LIN {X -0.269,Y -575.719,Z 1184.977,A 0.000,B 0.000,C 90.000,E1 31.799} C_DIS
LIN {X 0.203,Y -573.633,Z 1184.974,A 0.000,B 0.000,C 90.000,E1 31.209} C_DIS
LIN {X 0.086,Y -570.715,Z 1184.970,A 0.000,B 0.000,C 90.000,E1 30.541} C_DIS
LIN {X -0.150,Y -566.853,Z 1184.965,A 0.000,B 0.000,C 90.000,E1 29.745} C_DIS
LIN {X 0.163,Y -563.307,Z 1184.961,A 0.000,B 0.000,C 90.000,E1 29.027} C_DIS
LIN {X -0.358,Y -557.017,Z 1184.955,A 0.000,B 0.000,C 90.000,E1 27.975} C_DIS
LIN {X -0.139,Y -552.755,Z 1184.951,A 0.000,B 0.000,C 90.000,E1 27.257} C_DIS
LIN {X 0.150,Y -549.096,Z 1184.948,A 0.000,B 0.000,C 90.000,E1 26.668} C_DIS
LIN {X 0.138,Y -544.085,Z 1184.944,A 0.000,B 0.000,C 90.000,E1 25.976} C_DIS
LIN {X -0.009,Y -538.645,Z 1184.941,A 0.000,B 0.000,C 90.000,E1 25.283} C_DIS
LIN {X -0.197,Y -532.873,Z 1184.937,A 0.000,B 0.000,C 90.000,E1 24.591} C_DIS
LIN {X 0.108,Y -525.350,Z 1184.932,A 0.000,B 0.000,C 90.000,E1 23.695} C_DIS
LIN {X -0.102,Y -518.911,Z 1184.928,A 0.000,B 0.000,C 90.000,E1 23.003} C_DIS
LIN {X 0.115,Y -510.878,Z 1184.923,A 0.000,B 0.000,C 90.000,E1 22.153} C_DIS
LIN {X 0.130,Y -504.007,Z 1184.919,A 0.000,B 0.000,C 90.000,E1 21.461} C_DIS
LIN {X 0.176,Y -495.817,Z 1184.915,A 0.000,B 0.000,C 90.000,E1 20.663} C_DIS
LIN {X 0.012,Y -484.326,Z 1184.909,A 0.000,B 0.000,C 90.000,E1 19.631} C_DIS
LIN {X 0.204,Y -477.159,Z 1184.906,A 0.000,B 0.000,C 90.000,E1 18.960} C_DIS
LIN {X -0.109,Y -468.645,Z 1184.901,A 0.000,B 0.000,C 90.000,E1 18.236} C_DIS
LIN {X 0.094,Y -449.703,Z 1184.892,A 0.000,B 0.000,C 90.000,E1 16.496} C_DIS
LIN {X -0.072,Y -429.494,Z 1184.881,A 0.000,B 0.000,C 90.000,E1 14.537} C_DIS
LIN {X -0.024,Y -415.561,Z 1184.872,A 0.000,B 0.000,C 90.000,E1 13.008} C_DIS
LIN {X -0.139,Y -404.803,Z 1184.865,A 0.000,B 0.000,C 90.000,E1 11.715} C_DIS
LIN {X -0.011,Y -398.437,Z 1184.860,A 0.000,B 0.000,C 90.000,E1 10.838} C_DIS
LIN {X 0.029,Y -396.065,Z 1184.858,A 0.000,B 0.000,C 90.000,E1 10.433} C_DIS
LIN {X 0.074,Y -394.315,Z 1184.856,A 0.000,B 0.000,C 90.000,E1 10.074} C_DIS
LIN {X -0.105,Y -393.196,Z 1184.854,A 0.000,B 0.000,C 90.000,E1 9.792} C_DIS
LIN {X -0.142,Y -393.181,Z 1184.854,A 0.000,B 0.000,C 90.000,E1 9.792} C_DIS
LIN {X -0.065,Y -393.222,Z 1184.852,A 0.000,B 0.000,C 90.000,E1 9.443} C_DIS
LIN {X 0.077,Y -394.548,Z 1184.849,A 0.000,B 0.000,C 90.000,E1 8.803} C_DIS
LIN {X 0.005,Y -397.236,Z 1184.845,A 0.000,B 0.000,C 90.000,E1 8.106} C_DIS
LIN {X -0.079,Y -401.943,Z 1184.840,A 0.000,B 0.000,C 90.000,E1 7.239} C_DIS
LIN {X -0.159,Y -404.688,Z 1184.838,A 0.000,B 0.000,C 90.000,E1 6.891} C_DIS
LIN {X -0.150,Y -406.083,Z 1184.837,A 0.000,B 0.000,C 90.000,E1 6.720} C_DIS
LIN {X 0.070,Y -411.425,Z 1184.835,A 0.000,B 0.000,C 90.000,E1 6.201} C_DIS
LIN {X -0.139,Y -422.184,Z 1184.830,A 0.000,B 0.000,C 90.000,E1 5.391} C_DIS
LIN {X 0.231,Y -439.892,Z 1184.823,A 0.000,B 0.000,C 90.000,E1 4.012} C_DIS
LIN {X 0.057,Y -459.196,Z 1184.815,A 0.000,B 0.000,C 90.000,E1 2.636} C_DIS
LIN {X 0.128,Y -468.582,Z 1184.811,A 0.000,B 0.000,C 90.000,E1 1.949} C_DIS
LIN {X 0.139,Y -474.703,Z 1184.808,A 0.000,B 0.000,C 90.000,E1 1.489} C_DIS
LIN {X -0.061,Y -483.888,Z 1184.804,A 0.000,B 0.000,C 90.000,E1 0.802} C_DIS
LIN {X 0.030,Y -491.293,Z 1184.801,A 0.000,B 0.000,C 90.000,E1 0.172} C_DIS
LIN {X 0.065,Y -497.030,Z 1184.798,A 0.000,B 0.000,C 90.000,E1 359.656} C_DIS
LIN {X 0.152,Y -503.917,Z 1184.794,A 0.000,B 0.000,C 90.000,E1 358.969} C_DIS
LIN {X 0.242,Y -511.679,Z 1184.790,A 0.000,B 0.000,C 90.000,E1 358.108} C_DIS
LIN {X -0.203,Y -517.848,Z 1184.786,A 0.000,B 0.000,C 90.000,E1 357.421} C_DIS
LIN {X 0.215,Y -522.508,Z 1184.782,A 0.000,B 0.000,C 90.000,E1 356.788} C_DIS
LIN {X -0.165,Y -527.659,Z 1184.778,A 0.000,B 0.000,C 90.000,E1 356.102} C_DIS
LIN {X 0.060,Y -532.426,Z 1184.774,A 0.000,B 0.000,C 90.000,E1 355.355} C_DIS
LIN {X 0.070,Y -535.907,Z 1184.771,A 0.000,B 0.000,C 90.000,E1 354.780} C_DIS
LIN {X -0.108,Y -541.172,Z 1184.766,A 0.000,B 0.000,C 90.000,E1 353.799} C_DIS
LIN {X -0.034,Y -543.957,Z 1184.762,A 0.000,B 0.000,C 90.000,E1 353.223} C_DIS
LIN {X -0.132,Y -547.123,Z 1184.758,A 0.000,B 0.000,C 90.000,E1 352.527} C_DIS
LIN {X -0.279,Y -550.023,Z 1184.755,A 0.000,B 0.000,C 90.000,E1 351.837} C_DIS
LIN {X -0.041,Y -553.129,Z 1184.750,A 0.000,B 0.000,C 90.000,E1 350.971} C_DIS
LIN {X -0.225,Y -555.911,Z 1184.745,A 0.000,B 0.000,C 90.000,E1 350.151} C_DIS
LIN {X 0.212,Y -559.244,Z 1184.739,A 0.000,B 0.000,C 90.000,E1 348.993} C_DIS
LIN {X 0.097,Y -561.492,Z 1184.734,A 0.000,B 0.000,C 90.000,E1 348.173} C_DIS
LIN {X 0.167,Y -564.315,Z 1184.728,A 0.000,B 0.000,C 90.000,E1 347.061} C_DIS
LIN {X 0.025,Y -567.547,Z 1184.721,A 0.000,B 0.000,C 90.000,E1 345.700} C_DIS
LIN {X -0.058,Y -570.527,Z 1184.713,A 0.000,B 0.000,C 90.000,E1 344.338} C_DIS
LIN {X -0.281,Y -572.756,Z 1184.707,A 0.000,B 0.000,C 90.000,E1 343.268} C_DIS
LIN {X 0.055,Y -575.417,Z 1184.699,A 0.000,B 0.000,C 90.000,E1 341.873} C_DIS
LIN {X 0.075,Y -577.334,Z 1184.693,A 0.000,B 0.000,C 90.000,E1 340.786} C_DIS
LIN {X 0.115,Y -579.005,Z 1184.687,A 0.000,B 0.000,C 90.000,E1 339.699} C_DIS
LIN {X -0.163,Y -580.408,Z 1184.681,A 0.000,B 0.000,C 90.000,E1 338.646} C_DIS
LIN {X 0.264,Y -581.304,Z 1184.677,A 0.000,B 0.000,C 90.000,E1 337.794} C_DIS
LIN {X 0.015,Y -582.086,Z 1184.671,A 0.000,B 0.000,C 90.000,E1 336.741} C_DIS
LIN {X 0.142,Y -582.315,Z 1184.666,A 0.000,B 0.000,C 90.000,E1 335.921} C_DIS
LIN {X 0.275,Y -582.164,Z 1184.662,A 0.000,B 0.000,C 90.000,E1 335.101} C_DIS
LIN {X -0.119,Y -581.741,Z 1184.657,A 0.000,B 0.000,C 90.000,E1 334.332} C_DIS
LIN {X 0.008,Y -580.944,Z 1184.653,A 0.000,B 0.000,C 90.000,E1 333.512} C_DIS
LIN {X -0.261,Y -580.193,Z 1184.650,A 0.000,B 0.000,C 90.000,E1 332.999} C_DIS
LIN {X 0.108,Y -578.695,Z 1184.645,A 0.000,B 0.000,C 90.000,E1 332.153} C_DIS
LIN {X -0.321,Y -576.890,Z 1184.641,A 0.000,B 0.000,C 90.000,E1 331.385} C_DIS
LIN {X 0.163,Y -575.563,Z 1184.638,A 0.000,B 0.000,C 90.000,E1 330.795} C_DIS
LIN {X 0.137,Y -574.037,Z 1184.635,A 0.000,B 0.000,C 90.000,E1 330.255} C_DIS
LIN {X -0.183,Y -572.185,Z 1184.632,A 0.000,B 0.000,C 90.000,E1 329.744} C_DIS
LIN {X -0.059,Y -571.193,Z 1184.630,A 0.000,B 0.000,C 90.000,E1 329.459} C_DIS
LIN {X -0.108,Y -568.851,Z 1184.627,A 0.000,B 0.000,C 90.000,E1 328.918} C_DIS
LIN {X 0.106,Y -566.731,Z 1184.625,A 0.000,B 0.000,C 90.000,E1 328.486} C_DIS
LIN {X 0.018,Y -563.555,Z 1184.622,A 0.000,B 0.000,C 90.000,E1 327.946} C_DIS
LIN {X 0.106,Y -559.089,Z 1184.618,A 0.000,B 0.000,C 90.000,E1 327.248} C_DIS
LIN {X -0.033,Y -555.097,Z 1184.615,A 0.000,B 0.000,C 90.000,E1 326.707} C_DIS
LIN {X 0.108,Y -550.863,Z 1184.612,A 0.000,B 0.000,C 90.000,E1 326.135} C_DIS
LIN {X -0.220,Y -545.206,Z 1184.608,A 0.000,B 0.000,C 90.000,E1 325.468} C_DIS
LIN {X -0.265,Y -536.699,Z 1184.603,A 0.000,B 0.000,C 90.000,E1 324.482} C_DIS
LIN {X 0.122,Y -522.008,Z 1184.593,A 0.000,B 0.000,C 90.000,E1 322.763} C_DIS
LIN {X -0.102,Y -518.958,Z 1184.591,A 0.000,B 0.000,C 90.000,E1 322.351} C_DIS
LIN {X 0.324,Y -516.396,Z 1184.588,A 0.000,B 0.000,C 90.000,E1 321.823} C_DIS
LIN {X 0.010,Y -514.508,Z 1184.585,A 0.000,B 0.000,C 90.000,E1 321.251} C_DIS
LIN {X 0.113,Y -513.672,Z 1184.580,A 0.000,B 0.000,C 90.000,E1 320.356} C_DIS
LIN {X 0.035,Y -513.598,Z 1184.578,A 0.000,B 0.000,C 90.000,E1 320.070} C_DIS
LIN {X 0.125,Y -513.996,Z 1184.573,A 0.000,B 0.000,C 90.000,E1 319.175} C_DIS
LIN {X -0.168,Y -514.629,Z 1184.568,A 0.000,B 0.000,C 90.000,E1 318.324} C_DIS
LIN {X 0.079,Y -515.433,Z 1184.560,A 0.000,B 0.000,C 90.000,E1 316.824} C_DIS
LIN {X 0.163,Y -516.637,Z 1184.549,A 0.000,B 0.000,C 90.000,E1 314.757} C_DIS
LIN {X 0.077,Y -517.526,Z 1184.541,A 0.000,B 0.000,C 90.000,E1 313.299} C_DIS
LIN {X 0.236,Y -518.737,Z 1184.529,A 0.000,B 0.000,C 90.000,E1 311.229} C_DIS
LIN {X 0.147,Y -519.868,Z 1184.520,A 0.000,B 0.000,C 90.000,E1 309.483} C_DIS
LIN {X 0.150,Y -520.975,Z 1184.510,A 0.000,B 0.000,C 90.000,E1 307.729} C_DIS
LIN {X -0.141,Y -521.914,Z 1184.500,A 0.000,B 0.000,C 90.000,E1 306.011} C_DIS
LIN {X 0.052,Y -522.719,Z 1184.492,A 0.000,B 0.000,C 90.000,E1 304.532} C_DIS
LIN {X -0.084,Y -523.569,Z 1184.482,A 0.000,B 0.000,C 90.000,E1 302.801} C_DIS
LIN {X 0.002,Y -524.332,Z 1184.474,A 0.000,B 0.000,C 90.000,E1 301.337} C_DIS
LIN {X 0.029,Y -524.671,Z 1184.469,A 0.000,B 0.000,C 90.000,E1 300.463} C_DIS
LIN {X 0.138,Y -525.116,Z 1184.461,A 0.000,B 0.000,C 90.000,E1 298.999} C_DIS
LIN {X -0.007,Y -525.474,Z 1184.453,A 0.000,B 0.000,C 90.000,E1 297.564} C_DIS
LIN {X 0.082,Y -525.661,Z 1184.445,A 0.000,B 0.000,C 90.000,E1 296.104} C_DIS
LIN {X 0.180,Y -525.742,Z 1184.437,A 0.000,B 0.000,C 90.000,E1 294.643} C_DIS
LIN {X 0.062,Y -525.653,Z 1184.429,A 0.000,B 0.000,C 90.000,E1 293.206} C_DIS
LIN {X 0.106,Y -525.481,Z 1184.419,A 0.000,B 0.000,C 90.000,E1 291.461} C_DIS
LIN {X 0.269,Y -525.311,Z 1184.411,A 0.000,B 0.000,C 90.000,E1 289.993} C_DIS
LIN {X 0.089,Y -525.122,Z 1184.405,A 0.000,B 0.000,C 90.000,E1 288.852} C_DIS
LIN {X 0.077,Y -524.752,Z 1184.397,A 0.000,B 0.000,C 90.000,E1 287.402} C_DIS
LIN {X -0.099,Y -524.032,Z 1184.389,A 0.000,B 0.000,C 90.000,E1 285.969} C_DIS
LIN {X -0.149,Y -522.838,Z 1184.377,A 0.000,B 0.000,C 90.000,E1 283.939} C_DIS
LIN {X 0.007,Y -521.376,Z 1184.366,A 0.000,B 0.000,C 90.000,E1 281.883} C_DIS
LIN {X -0.078,Y -520.439,Z 1184.358,A 0.000,B 0.000,C 90.000,E1 280.433} C_DIS
LIN {X -0.081,Y -519.725,Z 1184.350,A 0.000,B 0.000,C 90.000,E1 278.973} C_DIS
LIN {X 0.244,Y -518.767,Z 1184.340,A 0.000,B 0.000,C 90.000,E1 277.182} C_DIS
LIN {X 0.049,Y -517.839,Z 1184.332,A 0.000,B 0.000,C 90.000,E1 275.739} C_DIS
LIN {X 0.131,Y -516.443,Z 1184.319,A 0.000,B 0.000,C 90.000,E1 273.383} C_DIS
LIN {X 0.140,Y -515.258,Z 1184.306,A 0.000,B 0.000,C 90.000,E1 271.031} C_DIS
LIN {X -0.140,Y -514.744,Z 1184.299,A 0.000,B 0.000,C 90.000,E1 269.885} C_DIS
LIN {X 0.011,Y -514.038,Z 1184.291,A 0.000,B 0.000,C 90.000,E1 268.396} C_DIS
LIN {X 0.158,Y -513.196,Z 1184.283,A 0.000,B 0.000,C 90.000,E1 266.906} C_DIS
LIN {X -0.193,Y -512.145,Z 1184.275,A 0.000,B 0.000,C 90.000,E1 265.469} C_DIS
LIN {X 0.043,Y -511.167,Z 1184.268,A 0.000,B 0.000,C 90.000,E1 264.261} C_DIS
LIN {X 0.218,Y -509.835,Z 1184.260,A 0.000,B 0.000,C 90.000,E1 262.761} C_DIS
LIN {X 0.221,Y -507.714,Z 1184.247,A 0.000,B 0.000,C 90.000,E1 260.387} C_DIS
LIN {X -0.110,Y -505.962,Z 1184.235,A 0.000,B 0.000,C 90.000,E1 258.342} C_DIS
LIN {X 0.057,Y -504.422,Z 1184.225,A 0.000,B 0.000,C 90.000,E1 256.533} C_DIS
LIN {X -0.007,Y -503.668,Z 1184.220,A 0.000,B 0.000,C 90.000,E1 255.644} C_DIS
LIN {X -0.080,Y -502.414,Z 1184.212,A 0.000,B 0.000,C 90.000,E1 254.157} C_DIS
LIN {X -0.045,Y -500.795,Z 1184.200,A 0.000,B 0.000,C 90.000,E1 252.054} C_DIS
LIN {X 0.041,Y -499.255,Z 1184.190,A 0.000,B 0.000,C 90.000,E1 250.242} C_DIS
LIN {X 0.189,Y -497.865,Z 1184.182,A 0.000,B 0.000,C 90.000,E1 248.720} C_DIS
LIN {X 0.084,Y -496.100,Z 1184.172,A 0.000,B 0.000,C 90.000,E1 246.922} C_DIS
LIN {X -0.162,Y -494.938,Z 1184.165,A 0.000,B 0.000,C 90.000,E1 245.741} C_DIS
LIN {X 0.031,Y -493.224,Z 1184.157,A 0.000,B 0.000,C 90.000,E1 244.204} C_DIS
LIN {X -0.054,Y -491.803,Z 1184.150,A 0.000,B 0.000,C 90.000,E1 242.999} C_DIS
LIN {X -0.106,Y -489.424,Z 1184.140,A 0.000,B 0.000,C 90.000,E1 241.179} C_DIS
LIN {X -0.033,Y -487.848,Z 1184.133,A 0.000,B 0.000,C 90.000,E1 239.950} C_DIS
LIN {X 0.067,Y -485.806,Z 1184.125,A 0.000,B 0.000,C 90.000,E1 238.408} C_DIS
LIN {X -0.279,Y -483.699,Z 1184.116,A 0.000,B 0.000,C 90.000,E1 236.914} C_DIS
LIN {X 0.295,Y -480.772,Z 1184.104,A 0.000,B 0.000,C 90.000,E1 234.689} C_DIS
LIN {X -0.078,Y -479.145,Z 1184.097,A 0.000,B 0.000,C 90.000,E1 233.497} C_DIS
LIN {X 0.079,Y -476.657,Z 1184.087,A 0.000,B 0.000,C 90.000,E1 231.618} C_DIS
LIN {X 0.015,Y -474.694,Z 1184.078,A 0.000,B 0.000,C 90.000,E1 230.070} C_DIS
LIN {X -0.137,Y -472.707,Z 1184.070,A 0.000,B 0.000,C 90.000,E1 228.528} C_DIS
LIN {X 0.082,Y -471.849,Z 1184.066,A 0.000,B 0.000,C 90.000,E1 227.877} C_DIS
LIN {X 0.003,Y -467.254,Z 1184.047,A 0.000,B 0.000,C 90.000,E1 224.433} C_DIS
LIN {X 0.157,Y -464.953,Z 1184.035,A 0.000,B 0.000,C 90.000,E1 222.204} C_DIS
LIN {X -0.172,Y -463.095,Z 1184.010,A 0.000,B 0.000,C 90.000,E1 217.810} C_DIS
LIN {X -0.268,Y -463.009,Z 1184.005,A 0.000,B 0.000,C 90.000,E1 216.870} C_DIS
LIN {X 0.030,Y -462.884,Z 1183.992,A 0.000,B 0.000,C 90.000,E1 214.612} C_DIS
LIN {X -0.057,Y -463.639,Z 1183.978,A 0.000,B 0.000,C 90.000,E1 212.084} C_DIS
LIN {X -0.248,Y -465.015,Z 1183.968,A 0.000,B 0.000,C 90.000,E1 210.207} C_DIS
LIN {X -0.010,Y -467.601,Z 1183.952,A 0.000,B 0.000,C 90.000,E1 207.334} C_DIS
LIN {X -0.234,Y -474.700,Z 1183.922,A 0.000,B 0.000,C 90.000,E1 202.025} C_DIS
LIN {X 0.287,Y -482.358,Z 1183.901,A 0.000,B 0.000,C 90.000,E1 198.236} C_DIS
LIN {X -0.133,Y -493.316,Z 1183.879,A 0.000,B 0.000,C 90.000,E1 194.300} C_DIS
LIN {X -0.074,Y -499.996,Z 1183.868,A 0.000,B 0.000,C 90.000,E1 192.175} C_DIS
LIN {X 0.000,Y -505.831,Z 1183.858,A 0.000,B 0.000,C 90.000,E1 190.366} C_DIS
LIN {X 0.124,Y -511.908,Z 1183.848,A 0.000,B 0.000,C 90.000,E1 188.568} C_DIS
LIN {X -0.175,Y -516.997,Z 1183.839,A 0.000,B 0.000,C 90.000,E1 187.125} C_DIS
LIN {X 0.138,Y -521.938,Z 1183.831,A 0.000,B 0.000,C 90.000,E1 185.625} C_DIS
LIN {X -0.063,Y -528.889,Z 1183.820,A 0.000,B 0.000,C 90.000,E1 183.612} C_DIS
LIN {X -0.138,Y -533.797,Z 1183.812,A 0.000,B 0.000,C 90.000,E1 182.178} C_DIS
LIN {X -0.132,Y -537.755,Z 1183.806,A 0.000,B 0.000,C 90.000,E1 181.031} C_DIS
LIN {X -0.006,Y -544.608,Z 1183.795,A 0.000,B 0.000,C 90.000,E1 179.026} C_DIS
LIN {X 0.206,Y -549.498,Z 1183.787,A 0.000,B 0.000,C 90.000,E1 177.593} C_DIS
LIN {X -0.045,Y -554.277,Z 1183.779,A 0.000,B 0.000,C 90.000,E1 176.216} C_DIS
LIN {X -0.181,Y -559.046,Z 1183.771,A 0.000,B 0.000,C 90.000,E1 174.837} C_DIS
LIN {X 0.067,Y -565.560,Z 1183.760,A 0.000,B 0.000,C 90.000,E1 172.875} C_DIS
LIN {X 0.196,Y -570.165,Z 1183.753,A 0.000,B 0.000,C 90.000,E1 171.489} C_DIS
LIN {X -0.274,Y -573.811,Z 1183.747,A 0.000,B 0.000,C 90.000,E1 170.443} C_DIS
LIN {X 0.080,Y -578.337,Z 1183.739,A 0.000,B 0.000,C 90.000,E1 169.050} C_DIS
LIN {X 0.289,Y -583.650,Z 1183.730,A 0.000,B 0.000,C 90.000,E1 167.409} C_DIS
LIN {X -0.214,Y -588.094,Z 1183.723,A 0.000,B 0.000,C 90.000,E1 166.117} C_DIS
LIN {X 0.069,Y -592.417,Z 1183.715,A 0.000,B 0.000,C 90.000,E1 164.755} C_DIS
LIN {X 0.298,Y -597.572,Z 1183.707,A 0.000,B 0.000,C 90.000,E1 163.142} C_DIS
LIN {X -0.123,Y -600.956,Z 1183.701,A 0.000,B 0.000,C 90.000,E1 162.127} C_DIS
LIN {X 0.256,Y -604.285,Z 1183.695,A 0.000,B 0.000,C 90.000,E1 161.040} C_DIS
LIN {X 0.043,Y -608.346,Z 1183.688,A 0.000,B 0.000,C 90.000,E1 159.752} C_DIS
LIN {X -0.049,Y -611.504,Z 1183.682,A 0.000,B 0.000,C 90.000,E1 158.720} C_DIS
LIN {X 0.088,Y -615.385,Z 1183.675,A 0.000,B 0.000,C 90.000,E1 157.411} C_DIS
LIN {X 0.317,Y -618.494,Z 1183.669,A 0.000,B 0.000,C 90.000,E1 156.357} C_DIS
LIN {X 0.016,Y -621.525,Z 1183.663,A 0.000,B 0.000,C 90.000,E1 155.357} C_DIS
LIN {X 0.034,Y -625.811,Z 1183.655,A 0.000,B 0.000,C 90.000,E1 153.819} C_DIS
LIN {X 0.122,Y -629.295,Z 1183.648,A 0.000,B 0.000,C 90.000,E1 152.538} C_DIS
LIN {X 0.259,Y -632.697,Z 1183.641,A 0.000,B 0.000,C 90.000,E1 151.257} C_DIS
LIN {X 0.157,Y -635.267,Z 1183.635,A 0.000,B 0.000,C 90.000,E1 150.255} C_DIS
LIN {X -0.229,Y -637.787,Z 1183.629,A 0.000,B 0.000,C 90.000,E1 149.282} C_DIS
LIN {X 0.122,Y -640.675,Z 1183.622,A 0.000,B 0.000,C 90.000,E1 147.995} C_DIS
LIN {X 0.123,Y -642.870,Z 1183.617,A 0.000,B 0.000,C 90.000,E1 146.993} C_DIS
LIN {X -0.034,Y -644.980,Z 1183.611,A 0.000,B 0.000,C 90.000,E1 146.008} C_DIS
LIN {X -0.102,Y -647.422,Z 1183.604,A 0.000,B 0.000,C 90.000,E1 144.769} C_DIS
LIN {X 0.154,Y -650.152,Z 1183.596,A 0.000,B 0.000,C 90.000,E1 143.256} C_DIS
LIN {X 0.072,Y -652.762,Z 1183.588,A 0.000,B 0.000,C 90.000,E1 141.778} C_DIS
LIN {X -0.180,Y -656.501,Z 1183.577,A 0.000,B 0.000,C 90.000,E1 139.828} C_DIS
LIN {X -0.265,Y -658.488,Z 1183.571,A 0.000,B 0.000,C 90.000,E1 138.852} C_DIS
LIN {X 0.090,Y -661.172,Z 1183.564,A 0.000,B 0.000,C 90.000,E1 137.595} C_DIS
LIN {X 0.031,Y -664.270,Z 1183.556,A 0.000,B 0.000,C 90.000,E1 136.134} C_DIS
LIN {X 0.011,Y -668.494,Z 1183.546,A 0.000,B 0.000,C 90.000,E1 134.190} C_DIS
LIN {X 0.162,Y -674.179,Z 1183.532,A 0.000,B 0.000,C 90.000,E1 131.757} C_DIS
LIN {X -0.441,Y -679.395,Z 1183.520,A 0.000,B 0.000,C 90.000,E1 129.644} C_DIS
LIN {X -0.060,Y -682.953,Z 1183.512,A 0.000,B 0.000,C 90.000,E1 128.177} C_DIS
LIN {X -0.366,Y -687.741,Z 1183.502,A 0.000,B 0.000,C 90.000,E1 126.297} C_DIS
LIN {X -0.285,Y -690.679,Z 1183.495,A 0.000,B 0.000,C 90.000,E1 125.105} C_DIS
LIN {X -0.158,Y -693.453,Z 1183.488,A 0.000,B 0.000,C 90.000,E1 123.913} C_DIS
LIN {X -0.027,Y -695.531,Z 1183.483,A 0.000,B 0.000,C 90.000,E1 122.959} C_DIS
LIN {X -0.213,Y -698.049,Z 1183.477,A 0.000,B 0.000,C 90.000,E1 121.799} C_DIS
LIN {X 0.232,Y -700.396,Z 1183.470,A 0.000,B 0.000,C 90.000,E1 120.590} C_DIS
LIN {X -0.249,Y -702.441,Z 1183.464,A 0.000,B 0.000,C 90.000,E1 119.461} C_DIS
LIN {X 0.245,Y -703.928,Z 1183.458,A 0.000,B 0.000,C 90.000,E1 118.487} C_DIS
LIN {X -0.188,Y -705.309,Z 1183.453,A 0.000,B 0.000,C 90.000,E1 117.590} C_DIS
LIN {X 0.056,Y -706.086,Z 1183.449,A 0.000,B 0.000,C 90.000,E1 116.873} C_DIS
LIN {X -0.351,Y -706.587,Z 1183.444,A 0.000,B 0.000,C 90.000,E1 115.976} C_DIS
LIN {X 0.238,Y -706.682,Z 1183.442,A 0.000,B 0.000,C 90.000,E1 115.463} C_DIS
LIN {X 0.179,Y -706.508,Z 1183.438,A 0.000,B 0.000,C 90.000,E1 114.771} C_DIS
LIN {X -0.171,Y -706.409,Z 1183.436,A 0.000,B 0.000,C 90.000,E1 114.567} C_DIS
LIN {X 0.120,Y -705.564,Z 1183.434,A 0.000,B 0.000,C 90.000,E1 114.079} C_DIS
LIN {X 0.410,Y -704.995,Z 1183.433,A 0.000,B 0.000,C 90.000,E1 113.823} C_DIS
LIN {X 0.052,Y -702.907,Z 1183.430,A 0.000,B 0.000,C 90.000,E1 113.387} C_DIS
LIN {X 0.190,Y -702.299,Z 1183.429,A 0.000,B 0.000,C 90.000,E1 113.259} C_DIS
LIN {X 0.053,Y -701.383,Z 1183.429,A 0.000,B 0.000,C 90.000,E1 113.153} C_DIS
LIN {X 0.035,Y -696.336,Z 1183.426,A 0.000,B 0.000,C 90.000,E1 112.695} C_DIS
LIN {X -0.031,Y -694.686,Z 1183.426,A 0.000,B 0.000,C 90.000,E1 112.589} C_DIS
LIN {X 0.171,Y -691.695,Z 1183.425,A 0.000,B 0.000,C 90.000,E1 112.461} C_DIS
LIN {X 0.102,Y -685.305,Z 1183.424,A 0.000,B 0.000,C 90.000,E1 112.280} C_DIS
LIN {X -0.112,Y -683.759,Z 1183.424,A 0.000,B 0.000,C 90.000,E1 112.280} C_DIS
LIN {X -0.109,Y -677.261,Z 1183.424,A 0.000,B 0.000,C 90.000,E1 112.259} C_DIS
LIN {X -0.142,Y -606.123,Z 1183.424,A 0.000,B 0.000,C 90.000,E1 112.259} C_DIS
LIN {X -0.123,Y -601.588,Z 1183.422,A 0.000,B 0.000,C 90.000,E1 111.950} C_DIS
LIN {X -0.165,Y -590.164,Z 1183.417,A 0.000,B 0.000,C 90.000,E1 111.025} C_DIS
LIN {X -0.077,Y -578.973,Z 1183.412,A 0.000,B 0.000,C 90.000,E1 110.120} C_DIS
LIN {X -0.012,Y -569.965,Z 1183.408,A 0.000,B 0.000,C 90.000,E1 109.450} C_DIS
LIN {X 0.012,Y -556.759,Z 1183.403,A 0.000,B 0.000,C 90.000,E1 108.489} C_DIS
LIN {X 0.021,Y -553.886,Z 1183.401,A 0.000,B 0.000,C 90.000,E1 108.181} C_DIS
LIN {X -0.107,Y -553.394,Z 1183.401,A 0.000,B 0.000,C 90.000,E1 108.127} C_DIS
LIN {X 0.212,Y -552.038,Z 1183.399,A 0.000,B 0.000,C 90.000,E1 107.819} C_DIS
LIN {X 0.187,Y -551.203,Z 1183.397,A 0.000,B 0.000,C 90.000,E1 107.402} C_DIS
LIN {X 0.026,Y -550.969,Z 1183.394,A 0.000,B 0.000,C 90.000,E1 106.858} C_DIS
LIN {X -0.036,Y -551.484,Z 1183.389,A 0.000,B 0.000,C 90.000,E1 106.024} C_DIS
LIN {X -0.146,Y -552.999,Z 1183.380,A 0.000,B 0.000,C 90.000,E1 104.356} C_DIS
LIN {X -0.122,Y -554.806,Z 1183.367,A 0.000,B 0.000,C 90.000,E1 102.119} C_DIS
LIN {X 0.144,Y -556.784,Z 1183.356,A 0.000,B 0.000,C 90.000,E1 100.141} C_DIS
LIN {X 0.188,Y -558.293,Z 1183.349,A 0.000,B 0.000,C 90.000,E1 98.746} C_DIS
LIN {X 0.251,Y -559.627,Z 1183.341,A 0.000,B 0.000,C 90.000,E1 97.352} C_DIS
LIN {X 0.117,Y -560.543,Z 1183.335,A 0.000,B 0.000,C 90.000,E1 96.258} C_DIS
LIN {X 0.218,Y -561.694,Z 1183.326,A 0.000,B 0.000,C 90.000,E1 94.588} C_DIS
LIN {X -0.268,Y -562.787,Z 1183.316,A 0.000,B 0.000,C 90.000,E1 92.980} C_DIS
LIN {X -0.092,Y -564.228,Z 1183.306,A 0.000,B 0.000,C 90.000,E1 91.031} C_DIS
LIN {X 0.001,Y -565.456,Z 1183.297,A 0.000,B 0.000,C 90.000,E1 89.370} C_DIS
LIN {X 0.133,Y -566.581,Z 1183.287,A 0.000,B 0.000,C 90.000,E1 87.707} C_DIS
LIN {X -0.282,Y -567.721,Z 1183.278,A 0.000,B 0.000,C 90.000,E1 86.102} C_DIS
LIN {X -0.194,Y -568.668,Z 1183.271,A 0.000,B 0.000,C 90.000,E1 84.723} C_DIS
LIN {X 0.080,Y -569.811,Z 1183.261,A 0.000,B 0.000,C 90.000,E1 83.053} C_DIS
LIN {X -0.302,Y -570.711,Z 1183.254,A 0.000,B 0.000,C 90.000,E1 81.724} C_DIS
LIN {X -0.210,Y -571.384,Z 1183.248,A 0.000,B 0.000,C 90.000,E1 80.622} C_DIS
LIN {X 0.188,Y -572.174,Z 1183.240,A 0.000,B 0.000,C 90.000,E1 79.218} C_DIS
LIN {X -0.235,Y -573.206,Z 1183.230,A 0.000,B 0.000,C 90.000,E1 77.353} C_DIS
LIN {X -0.031,Y -574.064,Z 1183.221,A 0.000,B 0.000,C 90.000,E1 75.700} C_DIS
LIN {X 0.187,Y -574.886,Z 1183.212,A 0.000,B 0.000,C 90.000,E1 74.047} C_DIS
LIN {X -0.158,Y -576.247,Z 1183.198,A 0.000,B 0.000,C 90.000,E1 71.638} C_DIS
LIN {X 0.257,Y -577.413,Z 1183.187,A 0.000,B 0.000,C 90.000,E1 69.699} C_DIS
LIN {X 0.209,Y -579.237,Z 1183.175,A 0.000,B 0.000,C 90.000,E1 67.539} C_DIS
LIN {X 0.185,Y -580.912,Z 1183.166,A 0.000,B 0.000,C 90.000,E1 65.921} C_DIS
LIN {X 0.297,Y -582.639,Z 1183.156,A 0.000,B 0.000,C 90.000,E1 64.024} C_DIS
LIN {X 0.189,Y -584.506,Z 1183.146,A 0.000,B 0.000,C 90.000,E1 62.153} C_DIS
LIN {X -0.271,Y -585.991,Z 1183.136,A 0.000,B 0.000,C 90.000,E1 60.589} C_DIS
LIN {X 0.087,Y -587.390,Z 1183.128,A 0.000,B 0.000,C 90.000,E1 58.948} C_DIS
LIN {X 0.204,Y -588.233,Z 1183.122,A 0.000,B 0.000,C 90.000,E1 57.867} C_DIS
LIN {X 0.037,Y -589.178,Z 1183.114,A 0.000,B 0.000,C 90.000,E1 56.548} C_DIS
LIN {X -0.105,Y -590.148,Z 1183.107,A 0.000,B 0.000,C 90.000,E1 55.229} C_DIS
LIN {X 0.036,Y -590.900,Z 1183.101,A 0.000,B 0.000,C 90.000,E1 54.149} C_DIS
LIN {X 0.186,Y -591.535,Z 1183.096,A 0.000,B 0.000,C 90.000,E1 53.336} C_DIS
LIN {X -0.025,Y -593.012,Z 1183.083,A 0.000,B 0.000,C 90.000,E1 50.964} C_DIS
LIN {X 0.129,Y -593.608,Z 1183.076,A 0.000,B 0.000,C 90.000,E1 49.622} C_DIS
LIN {X 0.055,Y -594.283,Z 1183.067,A 0.000,B 0.000,C 90.000,E1 48.038} C_DIS
LIN {X -0.028,Y -594.459,Z 1183.061,A 0.000,B 0.000,C 90.000,E1 46.986} C_DIS
LIN {X -0.122,Y -594.491,Z 1183.052,A 0.000,B 0.000,C 90.000,E1 45.405} C_DIS
LIN {X -0.189,Y -594.320,Z 1183.046,A 0.000,B 0.000,C 90.000,E1 44.352} C_DIS
LIN {X -0.033,Y -594.046,Z 1183.042,A 0.000,B 0.000,C 90.000,E1 43.542} C_DIS
LIN {X -0.290,Y -593.608,Z 1183.037,A 0.000,B 0.000,C 90.000,E1 42.771} C_DIS
LIN {X -0.181,Y -592.733,Z 1183.030,A 0.000,B 0.000,C 90.000,E1 41.434} C_DIS
LIN {X -0.003,Y -592.182,Z 1183.026,A 0.000,B 0.000,C 90.000,E1 40.620} C_DIS
LIN {X 0.135,Y -590.914,Z 1183.018,A 0.000,B 0.000,C 90.000,E1 39.277} C_DIS
LIN {X 0.041,Y -589.797,Z 1183.012,A 0.000,B 0.000,C 90.000,E1 38.222} C_DIS
LIN {X 0.088,Y -589.128,Z 1183.009,A 0.000,B 0.000,C 90.000,E1 37.684} C_DIS
LIN {X -0.196,Y -587.049,Z 1183.002,A 0.000,B 0.000,C 90.000,E1 36.377} C_DIS
LIN {X -0.240,Y -585.137,Z 1182.996,A 0.000,B 0.000,C 90.000,E1 35.311} C_DIS
LIN {X 0.132,Y -583.973,Z 1182.993,A 0.000,B 0.000,C 90.000,E1 34.739} C_DIS
LIN {X -0.293,Y -581.353,Z 1182.987,A 0.000,B 0.000,C 90.000,E1 33.706} C_DIS
LIN {X -0.264,Y -578.121,Z 1182.981,A 0.000,B 0.000,C 90.000,E1 32.625} C_DIS
LIN {X -0.117,Y -575.306,Z 1182.977,A 0.000,B 0.000,C 90.000,E1 31.799} C_DIS
LIN {X -0.140,Y -573.231,Z 1182.974,A 0.000,B 0.000,C 90.000,E1 31.258} C_DIS
LIN {X -0.262,Y -570.273,Z 1182.970,A 0.000,B 0.000,C 90.000,E1 30.590} C_DIS
LIN {X -0.102,Y -565.727,Z 1182.964,A 0.000,B 0.000,C 90.000,E1 29.617} C_DIS
LIN {X -0.293,Y -562.104,Z 1182.961,A 0.000,B 0.000,C 90.000,E1 28.949} C_DIS
LIN {X -0.337,Y -555.728,Z 1182.955,A 0.000,B 0.000,C 90.000,E1 27.847} C_DIS
LIN {X -0.130,Y -551.354,Z 1182.951,A 0.000,B 0.000,C 90.000,E1 27.129} C_DIS
LIN {X 0.019,Y -548.594,Z 1182.948,A 0.000,B 0.000,C 90.000,E1 26.693} C_DIS
LIN {X 0.048,Y -542.411,Z 1182.944,A 0.000,B 0.000,C 90.000,E1 25.848} C_DIS
LIN {X -0.091,Y -536.952,Z 1182.940,A 0.000,B 0.000,C 90.000,E1 25.155} C_DIS
LIN {X -0.296,Y -531.006,Z 1182.936,A 0.000,B 0.000,C 90.000,E1 24.463} C_DIS
LIN {X -0.154,Y -522.173,Z 1182.930,A 0.000,B 0.000,C 90.000,E1 23.439} C_DIS
LIN {X 0.256,Y -516.872,Z 1182.927,A 0.000,B 0.000,C 90.000,E1 22.823} C_DIS
LIN {X -0.042,Y -507.536,Z 1182.922,A 0.000,B 0.000,C 90.000,E1 21.897} C_DIS
LIN {X 0.071,Y -496.324,Z 1182.916,A 0.000,B 0.000,C 90.000,E1 20.791} C_DIS
LIN {X -0.159,Y -484.736,Z 1182.910,A 0.000,B 0.000,C 90.000,E1 19.758} C_DIS
LIN {X -0.108,Y -477.357,Z 1182.906,A 0.000,B 0.000,C 90.000,E1 19.087} C_DIS
LIN {X -0.174,Y -468.548,Z 1182.902,A 0.000,B 0.000,C 90.000,E1 18.308} C_DIS
LIN {X 0.130,Y -448.451,Z 1182.891,A 0.000,B 0.000,C 90.000,E1 16.441} C_DIS
LIN {X 0.090,Y -429.593,Z 1182.881,A 0.000,B 0.000,C 90.000,E1 14.592} C_DIS
LIN {X 0.036,Y -415.515,Z 1182.873,A 0.000,B 0.000,C 90.000,E1 13.063} C_DIS
LIN {X 0.179,Y -404.697,Z 1182.865,A 0.000,B 0.000,C 90.000,E1 11.715} C_DIS
LIN {X -0.167,Y -398.247,Z 1182.860,A 0.000,B 0.000,C 90.000,E1 10.894} C_DIS
LIN {X -0.158,Y -395.251,Z 1182.858,A 0.000,B 0.000,C 90.000,E1 10.366} C_DIS
LIN {X -0.205,Y -394.427,Z 1182.857,A 0.000,B 0.000,C 90.000,E1 10.197} C_DIS
LIN {X -0.115,Y -393.206,Z 1182.855,A 0.000,B 0.000,C 90.000,E1 9.849} C_DIS
LIN {X -0.153,Y -393.197,Z 1182.855,A 0.000,B 0.000,C 90.000,E1 9.849} C_DIS
LIN {X -0.067,Y -393.253,Z 1182.852,A 0.000,B 0.000,C 90.000,E1 9.443} C_DIS
LIN {X -0.096,Y -394.427,Z 1182.849,A 0.000,B 0.000,C 90.000,E1 8.916} C_DIS
LIN {X -0.135,Y -395.593,Z 1182.848,A 0.000,B 0.000,C 90.000,E1 8.568} C_DIS
LIN {X 0.180,Y -397.641,Z 1182.845,A 0.000,B 0.000,C 90.000,E1 7.992} C_DIS
LIN {X 0.102,Y -402.314,Z 1182.840,A 0.000,B 0.000,C 90.000,E1 7.125} C_DIS
LIN {X 0.107,Y -406.480,Z 1182.837,A 0.000,B 0.000,C 90.000,E1 6.606} C_DIS
LIN {X -0.058,Y -411.855,Z 1182.834,A 0.000,B 0.000,C 90.000,E1 6.144} C_DIS
LIN {X 0.021,Y -421.410,Z 1182.830,A 0.000,B 0.000,C 90.000,E1 5.391} C_DIS
LIN {X -0.100,Y -440.743,Z 1182.822,A 0.000,B 0.000,C 90.000,E1 3.955} C_DIS
LIN {X -0.102,Y -459.811,Z 1182.814,A 0.000,B 0.000,C 90.000,E1 2.579} C_DIS
LIN {X -0.050,Y -470.866,Z 1182.810,A 0.000,B 0.000,C 90.000,E1 1.776} C_DIS
LIN {X -0.212,Y -481.583,Z 1182.805,A 0.000,B 0.000,C 90.000,E1 0.974} C_DIS
LIN {X 0.078,Y -487.546,Z 1182.803,A 0.000,B 0.000,C 90.000,E1 0.458} C_DIS
LIN {X -0.140,Y -491.931,Z 1182.801,A 0.000,B 0.000,C 90.000,E1 0.115} C_DIS
LIN {X 0.064,Y -496.865,Z 1182.798,A 0.000,B 0.000,C 90.000,E1 359.656} C_DIS
LIN {X 0.164,Y -503.823,Z 1182.794,A 0.000,B 0.000,C 90.000,E1 358.969} C_DIS
LIN {X -0.190,Y -511.596,Z 1182.790,A 0.000,B 0.000,C 90.000,E1 358.165} C_DIS
LIN {X -0.092,Y -517.785,Z 1182.786,A 0.000,B 0.000,C 90.000,E1 357.421} C_DIS
LIN {X -0.160,Y -522.458,Z 1182.782,A 0.000,B 0.000,C 90.000,E1 356.846} C_DIS
LIN {X -0.265,Y -528.617,Z 1182.778,A 0.000,B 0.000,C 90.000,E1 355.988} C_DIS
LIN {X 0.243,Y -532.449,Z 1182.774,A 0.000,B 0.000,C 90.000,E1 355.355} C_DIS
LIN {X 0.254,Y -535.967,Z 1182.771,A 0.000,B 0.000,C 90.000,E1 354.780} C_DIS
LIN {X -0.191,Y -540.565,Z 1182.766,A 0.000,B 0.000,C 90.000,E1 353.970} C_DIS
LIN {X -0.120,Y -543.446,Z 1182.763,A 0.000,B 0.000,C 90.000,E1 353.394} C_DIS
LIN {X 0.251,Y -546.690,Z 1182.759,A 0.000,B 0.000,C 90.000,E1 352.648} C_DIS
LIN {X -0.084,Y -550.237,Z 1182.755,A 0.000,B 0.000,C 90.000,E1 351.837} C_DIS
LIN {X 0.157,Y -553.353,Z 1182.750,A 0.000,B 0.000,C 90.000,E1 350.971} C_DIS
LIN {X -0.025,Y -556.153,Z 1182.745,A 0.000,B 0.000,C 90.000,E1 350.151} C_DIS
LIN {X -0.132,Y -559.510,Z 1182.739,A 0.000,B 0.000,C 90.000,E1 349.050} C_DIS
LIN {X -0.091,Y -562.530,Z 1182.733,A 0.000,B 0.000,C 90.000,E1 347.937} C_DIS
LIN {X -0.007,Y -565.290,Z 1182.727,A 0.000,B 0.000,C 90.000,E1 346.825} C_DIS
LIN {X -0.131,Y -568.501,Z 1182.719,A 0.000,B 0.000,C 90.000,E1 345.463} C_DIS
LIN {X -0.200,Y -571.434,Z 1182.712,A 0.000,B 0.000,C 90.000,E1 344.102} C_DIS
LIN {X 0.303,Y -573.643,Z 1182.706,A 0.000,B 0.000,C 90.000,E1 342.960} C_DIS
LIN {X -0.064,Y -576.296,Z 1182.698,A 0.000,B 0.000,C 90.000,E1 341.638} C_DIS
LIN {X -0.037,Y -578.192,Z 1182.692,A 0.000,B 0.000,C 90.000,E1 340.550} C_DIS
LIN {X 0.214,Y -579.817,Z 1182.686,A 0.000,B 0.000,C 90.000,E1 339.444} C_DIS
LIN {X 0.098,Y -580.889,Z 1182.682,A 0.000,B 0.000,C 90.000,E1 338.646} C_DIS
LIN {X -0.150,Y -582.072,Z 1182.676,A 0.000,B 0.000,C 90.000,E1 337.592} C_DIS
LIN {X 0.153,Y -582.737,Z 1182.670,A 0.000,B 0.000,C 90.000,E1 336.485} C_DIS
LIN {X -0.110,Y -582.898,Z 1182.667,A 0.000,B 0.000,C 90.000,E1 335.973} C_DIS
LIN {X 0.161,Y -582.890,Z 1182.664,A 0.000,B 0.000,C 90.000,E1 335.409} C_DIS
LIN {X 0.302,Y -582.549,Z 1182.659,A 0.000,B 0.000,C 90.000,E1 334.588} C_DIS
LIN {X -0.086,Y -581.894,Z 1182.655,A 0.000,B 0.000,C 90.000,E1 333.819} C_DIS
LIN {X 0.173,Y -581.336,Z 1182.652,A 0.000,B 0.000,C 90.000,E1 333.256} C_DIS
LIN {X -0.229,Y -580.011,Z 1182.647,A 0.000,B 0.000,C 90.000,E1 332.487} C_DIS
LIN {X 0.139,Y -578.344,Z 1182.643,A 0.000,B 0.000,C 90.000,E1 331.641} C_DIS
LIN {X -0.019,Y -576.421,Z 1182.638,A 0.000,B 0.000,C 90.000,E1 330.845} C_DIS
LIN {X 0.307,Y -574.103,Z 1182.634,A 0.000,B 0.000,C 90.000,E1 329.999} C_DIS
LIN {X 0.108,Y -571.063,Z 1182.629,A 0.000,B 0.000,C 90.000,E1 329.203} C_DIS
LIN {X 0.143,Y -569.234,Z 1182.627,A 0.000,B 0.000,C 90.000,E1 328.791} C_DIS
LIN {X -0.126,Y -567.087,Z 1182.625,A 0.000,B 0.000,C 90.000,E1 328.408} C_DIS
LIN {X -0.007,Y -563.004,Z 1182.621,A 0.000,B 0.000,C 90.000,E1 327.709} C_DIS
LIN {X -0.009,Y -560.398,Z 1182.618,A 0.000,B 0.000,C 90.000,E1 327.296} C_DIS
LIN {X -0.361,Y -554.367,Z 1182.614,A 0.000,B 0.000,C 90.000,E1 326.501} C_DIS
LIN {X 0.356,Y -551.194,Z 1182.611,A 0.000,B 0.000,C 90.000,E1 326.008} C_DIS
LIN {X 0.159,Y -546.622,Z 1182.608,A 0.000,B 0.000,C 90.000,E1 325.468} C_DIS
LIN {X 0.125,Y -538.205,Z 1182.603,A 0.000,B 0.000,C 90.000,E1 324.482} C_DIS
LIN {X 0.344,Y -533.339,Z 1182.600,A 0.000,B 0.000,C 90.000,E1 323.909} C_DIS
LIN {X 0.168,Y -522.411,Z 1182.593,A 0.000,B 0.000,C 90.000,E1 322.683} C_DIS
LIN {X -0.012,Y -518.831,Z 1182.590,A 0.000,B 0.000,C 90.000,E1 322.190} C_DIS
LIN {X 0.067,Y -516.614,Z 1182.588,A 0.000,B 0.000,C 90.000,E1 321.743} C_DIS
LIN {X -0.063,Y -514.803,Z 1182.584,A 0.000,B 0.000,C 90.000,E1 321.170} C_DIS
LIN {X -0.117,Y -514.110,Z 1182.580,A 0.000,B 0.000,C 90.000,E1 320.436} C_DIS
LIN {X 0.059,Y -514.028,Z 1182.577,A 0.000,B 0.000,C 90.000,E1 319.828} C_DIS
LIN {X -0.049,Y -514.910,Z 1182.569,A 0.000,B 0.000,C 90.000,E1 318.366} C_DIS
LIN {X -0.224,Y -515.852,Z 1182.559,A 0.000,B 0.000,C 90.000,E1 316.620} C_DIS
LIN {X -0.050,Y -516.921,Z 1182.549,A 0.000,B 0.000,C 90.000,E1 314.838} C_DIS
LIN {X -0.131,Y -517.807,Z 1182.541,A 0.000,B 0.000,C 90.000,E1 313.380} C_DIS
LIN {X 0.036,Y -519.037,Z 1182.530,A 0.000,B 0.000,C 90.000,E1 311.310} C_DIS
LIN {X -0.100,Y -520.349,Z 1182.518,A 0.000,B 0.000,C 90.000,E1 309.277} C_DIS
LIN {X -0.034,Y -521.259,Z 1182.510,A 0.000,B 0.000,C 90.000,E1 307.810} C_DIS
LIN {X 0.063,Y -522.398,Z 1182.499,A 0.000,B 0.000,C 90.000,E1 305.758} C_DIS
LIN {X 0.231,Y -523.342,Z 1182.489,A 0.000,B 0.000,C 90.000,E1 303.992} C_DIS
LIN {X -0.219,Y -524.387,Z 1182.478,A 0.000,B 0.000,C 90.000,E1 302.005} C_DIS
LIN {X -0.109,Y -525.041,Z 1182.470,A 0.000,B 0.000,C 90.000,E1 300.541} C_DIS
LIN {X 0.012,Y -525.529,Z 1182.462,A 0.000,B 0.000,C 90.000,E1 299.077} C_DIS
LIN {X -0.120,Y -525.905,Z 1182.453,A 0.000,B 0.000,C 90.000,E1 297.641} C_DIS
LIN {X -0.018,Y -526.081,Z 1182.445,A 0.000,B 0.000,C 90.000,E1 296.181} C_DIS
LIN {X -0.074,Y -526.188,Z 1182.439,A 0.000,B 0.000,C 90.000,E1 295.027} C_DIS
LIN {X 0.029,Y -526.145,Z 1182.431,A 0.000,B 0.000,C 90.000,E1 293.567} C_DIS
LIN {X 0.054,Y -525.922,Z 1182.420,A 0.000,B 0.000,C 90.000,E1 291.535} C_DIS
LIN {X -0.092,Y -525.687,Z 1182.410,A 0.000,B 0.000,C 90.000,E1 289.812} C_DIS
LIN {X 0.064,Y -525.349,Z 1182.400,A 0.000,B 0.000,C 90.000,E1 288.055} C_DIS
LIN {X -0.271,Y -525.068,Z 1182.396,A 0.000,B 0.000,C 90.000,E1 287.221} C_DIS
LIN {X 0.055,Y -524.523,Z 1182.389,A 0.000,B 0.000,C 90.000,E1 286.024} C_DIS
LIN {X -0.123,Y -523.557,Z 1182.379,A 0.000,B 0.000,C 90.000,E1 284.300} C_DIS
LIN {X 0.037,Y -522.759,Z 1182.373,A 0.000,B 0.000,C 90.000,E1 283.119} C_DIS
LIN {X 0.096,Y -521.146,Z 1182.360,A 0.000,B 0.000,C 90.000,E1 280.782} C_DIS
LIN {X 0.104,Y -520.242,Z 1182.350,A 0.000,B 0.000,C 90.000,E1 279.029} C_DIS
LIN {X -0.078,Y -519.248,Z 1182.341,A 0.000,B 0.000,C 90.000,E1 277.296} C_DIS
LIN {X 0.179,Y -518.126,Z 1182.331,A 0.000,B 0.000,C 90.000,E1 275.511} C_DIS
LIN {X -0.105,Y -517.061,Z 1182.321,A 0.000,B 0.000,C 90.000,E1 273.784} C_DIS
LIN {X -0.014,Y -515.995,Z 1182.310,A 0.000,B 0.000,C 90.000,E1 271.718} C_DIS
LIN {X 0.161,Y -515.373,Z 1182.301,A 0.000,B 0.000,C 90.000,E1 270.229} C_DIS
LIN {X -0.262,Y -514.525,Z 1182.292,A 0.000,B 0.000,C 90.000,E1 268.511} C_DIS
LIN {X -0.105,Y -513.750,Z 1182.283,A 0.000,B 0.000,C 90.000,E1 267.020} C_DIS
LIN {X 0.151,Y -512.935,Z 1182.277,A 0.000,B 0.000,C 90.000,E1 265.812} C_DIS
LIN {X -0.153,Y -512.002,Z 1182.270,A 0.000,B 0.000,C 90.000,E1 264.666} C_DIS
LIN {X -0.008,Y -510.474,Z 1182.260,A 0.000,B 0.000,C 90.000,E1 262.875} C_DIS
LIN {X 0.021,Y -508.302,Z 1182.247,A 0.000,B 0.000,C 90.000,E1 260.500} C_DIS
LIN {X 0.055,Y -506.263,Z 1182.234,A 0.000,B 0.000,C 90.000,E1 258.117} C_DIS
LIN {X -0.156,Y -504.291,Z 1182.221,A 0.000,B 0.000,C 90.000,E1 255.755} C_DIS
LIN {X 0.129,Y -502.439,Z 1182.209,A 0.000,B 0.000,C 90.000,E1 253.630} C_DIS
LIN {X 0.256,Y -501.464,Z 1182.203,A 0.000,B 0.000,C 90.000,E1 252.417} C_DIS
LIN {X 0.240,Y -501.051,Z 1182.199,A 0.000,B 0.000,C 90.000,E1 251.819} C_DIS
LIN {X -0.145,Y -499.513,Z 1182.189,A 0.000,B 0.000,C 90.000,E1 250.061} C_DIS
LIN {X 0.008,Y -498.072,Z 1182.181,A 0.000,B 0.000,C 90.000,E1 248.539} C_DIS
LIN {X -0.152,Y -496.610,Z 1182.172,A 0.000,B 0.000,C 90.000,E1 247.050} C_DIS
LIN {X 0.264,Y -495.442,Z 1182.166,A 0.000,B 0.000,C 90.000,E1 245.793} C_DIS
LIN {X -0.189,Y -493.740,Z 1182.157,A 0.000,B 0.000,C 90.000,E1 244.332} C_DIS
LIN {X -0.010,Y -491.893,Z 1182.149,A 0.000,B 0.000,C 90.000,E1 242.794} C_DIS
LIN {X -0.046,Y -489.145,Z 1182.137,A 0.000,B 0.000,C 90.000,E1 240.667} C_DIS
LIN {X 0.070,Y -486.684,Z 1182.127,A 0.000,B 0.000,C 90.000,E1 238.820} C_DIS
LIN {X -0.002,Y -484.566,Z 1182.118,A 0.000,B 0.000,C 90.000,E1 237.296} C_DIS
LIN {X 0.147,Y -481.188,Z 1182.105,A 0.000,B 0.000,C 90.000,E1 234.815} C_DIS
LIN {X -0.023,Y -479.126,Z 1182.096,A 0.000,B 0.000,C 90.000,E1 233.290} C_DIS
LIN {X 0.129,Y -476.602,Z 1182.086,A 0.000,B 0.000,C 90.000,E1 231.412} C_DIS
LIN {X -0.062,Y -473.830,Z 1182.074,A 0.000,B 0.000,C 90.000,E1 229.256} C_DIS
LIN {X -0.008,Y -472.179,Z 1182.067,A 0.000,B 0.000,C 90.000,E1 228.000} C_DIS
LIN {X 0.195,Y -467.801,Z 1182.049,A 0.000,B 0.000,C 90.000,E1 224.838} C_DIS
LIN {X -0.227,Y -465.044,Z 1182.035,A 0.000,B 0.000,C 90.000,E1 222.366} C_DIS
LIN {X 0.008,Y -462.882,Z 1182.005,A 0.000,B 0.000,C 90.000,E1 216.950} C_DIS
LIN {X -0.175,Y -463.266,Z 1181.979,A 0.000,B 0.000,C 90.000,E1 212.212} C_DIS
LIN {X -0.236,Y -464.814,Z 1181.967,A 0.000,B 0.000,C 90.000,E1 210.001} C_DIS
LIN {X -0.158,Y -467.065,Z 1181.953,A 0.000,B 0.000,C 90.000,E1 207.462} C_DIS
LIN {X 0.053,Y -473.562,Z 1181.925,A 0.000,B 0.000,C 90.000,E1 202.408} C_DIS
LIN {X 0.078,Y -481.707,Z 1181.902,A 0.000,B 0.000,C 90.000,E1 198.362} C_DIS
LIN {X 0.236,Y -492.697,Z 1181.880,A 0.000,B 0.000,C 90.000,E1 194.356} C_DIS
LIN {X 0.095,Y -500.351,Z 1181.866,A 0.000,B 0.000,C 90.000,E1 191.951} C_DIS
LIN {X 0.192,Y -506.218,Z 1181.857,A 0.000,B 0.000,C 90.000,E1 190.141} C_DIS
LIN {X -0.053,Y -511.335,Z 1181.848,A 0.000,B 0.000,C 90.000,E1 188.681} C_DIS
LIN {X 0.120,Y -517.497,Z 1181.838,A 0.000,B 0.000,C 90.000,E1 186.891} C_DIS
LIN {X -0.143,Y -523.443,Z 1181.829,A 0.000,B 0.000,C 90.000,E1 185.163} C_DIS
LIN {X 0.209,Y -529.465,Z 1181.819,A 0.000,B 0.000,C 90.000,E1 183.383} C_DIS
LIN {X 0.162,Y -535.427,Z 1181.809,A 0.000,B 0.000,C 90.000,E1 181.661} C_DIS
LIN {X 0.208,Y -541.293,Z 1181.800,A 0.000,B 0.000,C 90.000,E1 179.943} C_DIS
LIN {X -0.231,Y -545.292,Z 1181.794,A 0.000,B 0.000,C 90.000,E1 178.854} C_DIS
LIN {X -0.011,Y -550.215,Z 1181.786,A 0.000,B 0.000,C 90.000,E1 177.421} C_DIS
LIN {X -0.254,Y -554.990,Z 1181.778,A 0.000,B 0.000,C 90.000,E1 176.045} C_DIS
LIN {X 0.103,Y -558.868,Z 1181.772,A 0.000,B 0.000,C 90.000,E1 174.894} C_DIS
LIN {X -0.210,Y -565.465,Z 1181.761,A 0.000,B 0.000,C 90.000,E1 172.989} C_DIS
LIN {X -0.081,Y -570.125,Z 1181.753,A 0.000,B 0.000,C 90.000,E1 171.602} C_DIS
LIN {X -0.250,Y -575.674,Z 1181.744,A 0.000,B 0.000,C 90.000,E1 169.982} C_DIS
LIN {X 0.025,Y -579.287,Z 1181.738,A 0.000,B 0.000,C 90.000,E1 168.870} C_DIS
LIN {X 0.023,Y -583.789,Z 1181.731,A 0.000,B 0.000,C 90.000,E1 167.521} C_DIS
LIN {X 0.099,Y -588.283,Z 1181.723,A 0.000,B 0.000,C 90.000,E1 166.172} C_DIS
LIN {X -0.181,Y -592.630,Z 1181.716,A 0.000,B 0.000,C 90.000,E1 164.866} C_DIS
LIN {X 0.185,Y -596.967,Z 1181.708,A 0.000,B 0.000,C 90.000,E1 163.504} C_DIS
LIN {X 0.220,Y -601.180,Z 1181.701,A 0.000,B 0.000,C 90.000,E1 162.181} C_DIS
LIN {X 0.124,Y -603.693,Z 1181.697,A 0.000,B 0.000,C 90.000,E1 161.402} C_DIS
LIN {X -0.101,Y -607.773,Z 1181.690,A 0.000,B 0.000,C 90.000,E1 160.115} C_DIS
LIN {X 0.322,Y -611.705,Z 1181.682,A 0.000,B 0.000,C 90.000,E1 158.773} C_DIS
LIN {X 0.204,Y -616.325,Z 1181.674,A 0.000,B 0.000,C 90.000,E1 157.230} C_DIS
LIN {X -0.107,Y -618.638,Z 1181.669,A 0.000,B 0.000,C 90.000,E1 156.485} C_DIS
LIN {X 0.150,Y -622.369,Z 1181.662,A 0.000,B 0.000,C 90.000,E1 155.177} C_DIS
LIN {X 0.180,Y -626.560,Z 1181.654,A 0.000,B 0.000,C 90.000,E1 153.640} C_DIS
LIN {X 0.251,Y -629.340,Z 1181.648,A 0.000,B 0.000,C 90.000,E1 152.615} C_DIS
LIN {X -0.139,Y -633.385,Z 1181.640,A 0.000,B 0.000,C 90.000,E1 151.129} C_DIS
LIN {X 0.279,Y -635.294,Z 1181.635,A 0.000,B 0.000,C 90.000,E1 150.333} C_DIS
LIN {X 0.215,Y -637.795,Z 1181.630,A 0.000,B 0.000,C 90.000,E1 149.331} C_DIS
LIN {X 0.187,Y -640.067,Z 1181.624,A 0.000,B 0.000,C 90.000,E1 148.329} C_DIS
LIN {X 0.184,Y -642.310,Z 1181.619,A 0.000,B 0.000,C 90.000,E1 147.327} C_DIS
LIN {X 0.073,Y -644.885,Z 1181.612,A 0.000,B 0.000,C 90.000,E1 146.087} C_DIS
LIN {X 0.000,Y -647.312,Z 1181.605,A 0.000,B 0.000,C 90.000,E1 144.848} C_DIS
LIN {X 0.250,Y -650.023,Z 1181.596,A 0.000,B 0.000,C 90.000,E1 143.336} C_DIS
LIN {X 0.120,Y -652.197,Z 1181.590,A 0.000,B 0.000,C 90.000,E1 142.110} C_DIS
LIN {X 0.019,Y -654.430,Z 1181.583,A 0.000,B 0.000,C 90.000,E1 140.884} C_DIS
LIN {X -0.147,Y -657.838,Z 1181.573,A 0.000,B 0.000,C 90.000,E1 139.175} C_DIS
LIN {X -0.300,Y -661.506,Z 1181.564,A 0.000,B 0.000,C 90.000,E1 137.472} C_DIS
LIN {X 0.094,Y -664.566,Z 1181.556,A 0.000,B 0.000,C 90.000,E1 135.972} C_DIS
LIN {X 0.083,Y -668.813,Z 1181.545,A 0.000,B 0.000,C 90.000,E1 134.028} C_DIS
LIN {X 0.225,Y -673.961,Z 1181.533,A 0.000,B 0.000,C 90.000,E1 131.838} C_DIS
LIN {X -0.382,Y -679.126,Z 1181.521,A 0.000,B 0.000,C 90.000,E1 129.725} C_DIS
LIN {X -0.003,Y -682.690,Z 1181.513,A 0.000,B 0.000,C 90.000,E1 128.257} C_DIS
LIN {X 0.065,Y -686.892,Z 1181.503,A 0.000,B 0.000,C 90.000,E1 126.583} C_DIS
LIN {X 0.134,Y -689.877,Z 1181.497,A 0.000,B 0.000,C 90.000,E1 125.391} C_DIS
LIN {X 0.253,Y -692.680,Z 1181.490,A 0.000,B 0.000,C 90.000,E1 124.199} C_DIS
LIN {X -0.202,Y -694.817,Z 1181.485,A 0.000,B 0.000,C 90.000,E1 123.293} C_DIS
LIN {X -0.155,Y -697.865,Z 1181.477,A 0.000,B 0.000,C 90.000,E1 121.878} C_DIS
LIN {X -0.048,Y -700.641,Z 1181.469,A 0.000,B 0.000,C 90.000,E1 120.463} C_DIS
LIN {X -0.188,Y -702.247,Z 1181.464,A 0.000,B 0.000,C 90.000,E1 119.539} C_DIS
LIN {X -0.310,Y -703.791,Z 1181.459,A 0.000,B 0.000,C 90.000,E1 118.615} C_DIS
LIN {X -0.133,Y -705.507,Z 1181.452,A 0.000,B 0.000,C 90.000,E1 117.436} C_DIS
LIN {X -0.212,Y -706.174,Z 1181.448,A 0.000,B 0.000,C 90.000,E1 116.744} C_DIS
LIN {X 0.018,Y -706.656,Z 1181.443,A 0.000,B 0.000,C 90.000,E1 115.796} C_DIS
LIN {X 0.264,Y -706.694,Z 1181.439,A 0.000,B 0.000,C 90.000,E1 115.079} C_DIS
LIN {X -0.088,Y -706.448,Z 1181.437,A 0.000,B 0.000,C 90.000,E1 114.643} C_DIS
LIN {X 0.204,Y -706.154,Z 1181.436,A 0.000,B 0.000,C 90.000,E1 114.387} C_DIS
LIN {X -0.148,Y -705.272,Z 1181.433,A 0.000,B 0.000,C 90.000,E1 113.951} C_DIS
LIN {X 0.142,Y -703.313,Z 1181.430,A 0.000,B 0.000,C 90.000,E1 113.462} C_DIS
LIN {X -0.222,Y -702.107,Z 1181.429,A 0.000,B 0.000,C 90.000,E1 113.259} C_DIS
LIN {X -0.083,Y -701.083,Z 1181.428,A 0.000,B 0.000,C 90.000,E1 113.131} C_DIS
LIN {X 0.370,Y -696.110,Z 1181.426,A 0.000,B 0.000,C 90.000,E1 112.642} C_DIS
LIN {X -0.349,Y -694.264,Z 1181.425,A 0.000,B 0.000,C 90.000,E1 112.589} C_DIS
LIN {X 0.107,Y -691.651,Z 1181.425,A 0.000,B 0.000,C 90.000,E1 112.461} C_DIS
LIN {X -0.070,Y -686.947,Z 1181.424,A 0.000,B 0.000,C 90.000,E1 112.333} C_DIS
LIN {X -0.061,Y -684.733,Z 1181.424,A 0.000,B 0.000,C 90.000,E1 112.280} C_DIS
LIN {X -0.164,Y -677.850,Z 1181.424,A 0.000,B 0.000,C 90.000,E1 112.259} C_DIS
LIN {X 0.354,Y -605.934,Z 1181.424,A 0.000,B 0.000,C 90.000,E1 112.206} C_DIS
LIN {X -0.049,Y -600.863,Z 1181.422,A 0.000,B 0.000,C 90.000,E1 111.897} C_DIS
LIN {X 0.257,Y -589.835,Z 1181.417,A 0.000,B 0.000,C 90.000,E1 110.972} C_DIS
LIN {X 0.100,Y -580.086,Z 1181.412,A 0.000,B 0.000,C 90.000,E1 110.194} C_DIS
LIN {X -0.149,Y -574.123,Z 1181.410,A 0.000,B 0.000,C 90.000,E1 109.758} C_DIS
LIN {X 0.010,Y -564.969,Z 1181.406,A 0.000,B 0.000,C 90.000,E1 109.087} C_DIS
LIN {X 0.110,Y -557.563,Z 1181.403,A 0.000,B 0.000,C 90.000,E1 108.544} C_DIS
LIN {X 0.156,Y -553.583,Z 1181.401,A 0.000,B 0.000,C 90.000,E1 108.181} C_DIS
LIN {X 0.050,Y -553.049,Z 1181.401,A 0.000,B 0.000,C 90.000,E1 108.127} C_DIS
LIN {X -0.153,Y -551.681,Z 1181.399,A 0.000,B 0.000,C 90.000,E1 107.873} C_DIS
LIN {X -0.248,Y -550.784,Z 1181.397,A 0.000,B 0.000,C 90.000,E1 107.457} C_DIS
LIN {X 0.115,Y -550.707,Z 1181.394,A 0.000,B 0.000,C 90.000,E1 106.858} C_DIS
LIN {X -0.063,Y -552.840,Z 1181.380,A 0.000,B 0.000,C 90.000,E1 104.356} C_DIS
LIN {X -0.169,Y -554.450,Z 1181.369,A 0.000,B 0.000,C 90.000,E1 102.411} C_DIS
LIN {X 0.220,Y -556.746,Z 1181.357,A 0.000,B 0.000,C 90.000,E1 100.141} C_DIS
LIN {X -0.288,Y -558.207,Z 1181.349,A 0.000,B 0.000,C 90.000,E1 98.803} C_DIS
LIN {X -0.230,Y -559.528,Z 1181.341,A 0.000,B 0.000,C 90.000,E1 97.409} C_DIS
LIN {X -0.230,Y -560.651,Z 1181.333,A 0.000,B 0.000,C 90.000,E1 96.024} C_DIS
LIN {X -0.180,Y -561.781,Z 1181.324,A 0.000,B 0.000,C 90.000,E1 94.359} C_DIS
LIN {X 0.103,Y -563.318,Z 1181.312,A 0.000,B 0.000,C 90.000,E1 92.121} C_DIS
LIN {X 0.083,Y -564.374,Z 1181.304,A 0.000,B 0.000,C 90.000,E1 90.745} C_DIS
LIN {X 0.180,Y -565.560,Z 1181.295,A 0.000,B 0.000,C 90.000,E1 89.083} C_DIS
LIN {X 0.083,Y -566.291,Z 1181.289,A 0.000,B 0.000,C 90.000,E1 87.993} C_DIS
LIN {X -0.027,Y -567.066,Z 1181.283,A 0.000,B 0.000,C 90.000,E1 86.906} C_DIS
LIN {X 0.161,Y -568.180,Z 1181.274,A 0.000,B 0.000,C 90.000,E1 85.241} C_DIS
LIN {X 0.031,Y -569.502,Z 1181.263,A 0.000,B 0.000,C 90.000,E1 83.337} C_DIS
LIN {X 0.217,Y -570.420,Z 1181.255,A 0.000,B 0.000,C 90.000,E1 81.951} C_DIS
LIN {X 0.313,Y -571.130,Z 1181.249,A 0.000,B 0.000,C 90.000,E1 80.849} C_DIS
LIN {X -0.235,Y -572.182,Z 1181.239,A 0.000,B 0.000,C 90.000,E1 78.993} C_DIS
LIN {X -0.185,Y -573.032,Z 1181.230,A 0.000,B 0.000,C 90.000,E1 77.353} C_DIS
LIN {X 0.015,Y -573.907,Z 1181.221,A 0.000,B 0.000,C 90.000,E1 75.700} C_DIS
LIN {X 0.035,Y -574.569,Z 1181.213,A 0.000,B 0.000,C 90.000,E1 74.338} C_DIS
LIN {X -0.129,Y -575.750,Z 1181.201,A 0.000,B 0.000,C 90.000,E1 72.181} C_DIS
LIN {X -0.099,Y -576.728,Z 1181.192,A 0.000,B 0.000,C 90.000,E1 70.550} C_DIS
LIN {X -0.236,Y -577.663,Z 1181.184,A 0.000,B 0.000,C 90.000,E1 69.209} C_DIS
LIN {X 0.091,Y -579.332,Z 1181.174,A 0.000,B 0.000,C 90.000,E1 67.283} C_DIS
LIN {X 0.213,Y -580.790,Z 1181.166,A 0.000,B 0.000,C 90.000,E1 65.921} C_DIS
LIN {X -0.202,Y -582.512,Z 1181.156,A 0.000,B 0.000,C 90.000,E1 64.076} C_DIS
LIN {X 0.211,Y -584.341,Z 1181.146,A 0.000,B 0.000,C 90.000,E1 62.153} C_DIS
LIN {X -0.254,Y -585.855,Z 1181.136,A 0.000,B 0.000,C 90.000,E1 60.589} C_DIS
LIN {X 0.102,Y -587.225,Z 1181.128,A 0.000,B 0.000,C 90.000,E1 58.948} C_DIS
LIN {X 0.217,Y -588.082,Z 1181.122,A 0.000,B 0.000,C 90.000,E1 57.867} C_DIS
LIN {X -0.082,Y -589.228,Z 1181.113,A 0.000,B 0.000,C 90.000,E1 56.294} C_DIS
LIN {X -0.026,Y -590.392,Z 1181.104,A 0.000,B 0.000,C 90.000,E1 54.689} C_DIS
LIN {X 0.189,Y -591.334,Z 1181.096,A 0.000,B 0.000,C 90.000,E1 53.336} C_DIS
LIN {X -0.241,Y -592.636,Z 1181.085,A 0.000,B 0.000,C 90.000,E1 51.251} C_DIS
LIN {X 0.152,Y -593.160,Z 1181.079,A 0.000,B 0.000,C 90.000,E1 50.150} C_DIS
LIN {X -0.141,Y -593.749,Z 1181.071,A 0.000,B 0.000,C 90.000,E1 48.852} C_DIS
LIN {X 0.043,Y -594.042,Z 1181.067,A 0.000,B 0.000,C 90.000,E1 48.038} C_DIS
LIN {X -0.042,Y -594.236,Z 1181.061,A 0.000,B 0.000,C 90.000,E1 46.986} C_DIS
LIN {X 0.087,Y -594.242,Z 1181.054,A 0.000,B 0.000,C 90.000,E1 45.648} C_DIS
LIN {X 0.017,Y -594.146,Z 1181.048,A 0.000,B 0.000,C 90.000,E1 44.595} C_DIS
LIN {X -0.058,Y -593.772,Z 1181.042,A 0.000,B 0.000,C 90.000,E1 43.542} C_DIS
LIN {X -0.317,Y -593.350,Z 1181.037,A 0.000,B 0.000,C 90.000,E1 42.771} C_DIS
LIN {X 0.232,Y -592.466,Z 1181.030,A 0.000,B 0.000,C 90.000,E1 41.391} C_DIS
LIN {X -0.038,Y -591.891,Z 1181.026,A 0.000,B 0.000,C 90.000,E1 40.620} C_DIS
LIN {X 0.096,Y -590.608,Z 1181.018,A 0.000,B 0.000,C 90.000,E1 39.277} C_DIS
LIN {X -0.003,Y -589.427,Z 1181.012,A 0.000,B 0.000,C 90.000,E1 38.222} C_DIS
LIN {X -0.222,Y -588.370,Z 1181.008,A 0.000,B 0.000,C 90.000,E1 37.443} C_DIS
LIN {X -0.248,Y -586.682,Z 1181.002,A 0.000,B 0.000,C 90.000,E1 36.377} C_DIS
LIN {X -0.297,Y -584.734,Z 1180.996,A 0.000,B 0.000,C 90.000,E1 35.311} C_DIS
LIN {X -0.078,Y -582.936,Z 1180.992,A 0.000,B 0.000,C 90.000,E1 34.485} C_DIS
LIN {X 0.126,Y -580.901,Z 1180.987,A 0.000,B 0.000,C 90.000,E1 33.658} C_DIS
LIN {X -0.024,Y -577.624,Z 1180.981,A 0.000,B 0.000,C 90.000,E1 32.594} C_DIS
LIN {X -0.194,Y -574.773,Z 1180.977,A 0.000,B 0.000,C 90.000,E1 31.799} C_DIS
LIN {X -0.219,Y -572.683,Z 1180.974,A 0.000,B 0.000,C 90.000,E1 31.258} C_DIS
LIN {X 0.146,Y -569.710,Z 1180.970,A 0.000,B 0.000,C 90.000,E1 30.541} C_DIS
LIN {X 0.087,Y -565.145,Z 1180.964,A 0.000,B 0.000,C 90.000,E1 29.589} C_DIS
LIN {X 0.277,Y -560.686,Z 1180.960,A 0.000,B 0.000,C 90.000,E1 28.743} C_DIS
LIN {X 0.311,Y -555.072,Z 1180.954,A 0.000,B 0.000,C 90.000,E1 27.769} C_DIS
LIN {X -0.237,Y -550.687,Z 1180.951,A 0.000,B 0.000,C 90.000,E1 27.129} C_DIS
LIN {X -0.091,Y -547.865,Z 1180.948,A 0.000,B 0.000,C 90.000,E1 26.693} C_DIS
LIN {X -0.215,Y -540.625,Z 1180.943,A 0.000,B 0.000,C 90.000,E1 25.720} C_DIS
LIN {X 0.096,Y -535.003,Z 1180.939,A 0.000,B 0.000,C 90.000,E1 24.975} C_DIS
LIN {X 0.239,Y -530.149,Z 1180.936,A 0.000,B 0.000,C 90.000,E1 24.387} C_DIS
LIN {X -0.176,Y -522.645,Z 1180.931,A 0.000,B 0.000,C 90.000,E1 23.567} C_DIS
LIN {X 0.221,Y -517.365,Z 1180.928,A 0.000,B 0.000,C 90.000,E1 22.950} C_DIS
LIN {X -0.168,Y -507.942,Z 1180.922,A 0.000,B 0.000,C 90.000,E1 22.025} C_DIS
LIN {X 0.098,Y -496.964,Z 1180.916,A 0.000,B 0.000,C 90.000,E1 20.918} C_DIS
LIN {X 0.061,Y -485.657,Z 1180.911,A 0.000,B 0.000,C 90.000,E1 19.885} C_DIS
LIN {X 0.128,Y -478.325,Z 1180.907,A 0.000,B 0.000,C 90.000,E1 19.214} C_DIS
LIN {X 0.041,Y -468.026,Z 1180.902,A 0.000,B 0.000,C 90.000,E1 18.308} C_DIS
LIN {X -0.070,Y -447.398,Z 1180.891,A 0.000,B 0.000,C 90.000,E1 16.441} C_DIS
LIN {X -0.027,Y -427.141,Z 1180.880,A 0.000,B 0.000,C 90.000,E1 14.426} C_DIS
LIN {X 0.114,Y -414.518,Z 1180.872,A 0.000,B 0.000,C 90.000,E1 13.008} C_DIS
LIN {X -0.042,Y -402.556,Z 1180.864,A 0.000,B 0.000,C 90.000,E1 11.535} C_DIS
LIN {X -0.050,Y -397.560,Z 1180.860,A 0.000,B 0.000,C 90.000,E1 10.838} C_DIS
LIN {X -0.044,Y -394.683,Z 1180.857,A 0.000,B 0.000,C 90.000,E1 10.310} C_DIS
LIN {X 0.031,Y -393.148,Z 1180.855,A 0.000,B 0.000,C 90.000,E1 9.849} C_DIS
LIN {X -0.007,Y -393.142,Z 1180.855,A 0.000,B 0.000,C 90.000,E1 9.849} C_DIS
LIN {X -0.112,Y -393.327,Z 1180.852,A 0.000,B 0.000,C 90.000,E1 9.443} C_DIS
LIN {X -0.141,Y -394.521,Z 1180.849,A 0.000,B 0.000,C 90.000,E1 8.916} C_DIS
LIN {X -0.181,Y -395.699,Z 1180.848,A 0.000,B 0.000,C 90.000,E1 8.568} C_DIS
LIN {X 0.135,Y -397.721,Z 1180.845,A 0.000,B 0.000,C 90.000,E1 7.992} C_DIS
LIN {X 0.194,Y -400.716,Z 1180.841,A 0.000,B 0.000,C 90.000,E1 7.409} C_DIS
LIN {X 0.128,Y -402.481,Z 1180.839,A 0.000,B 0.000,C 90.000,E1 7.068} C_DIS
LIN {X 0.094,Y -406.616,Z 1180.837,A 0.000,B 0.000,C 90.000,E1 6.549} C_DIS
LIN {X 0.025,Y -411.918,Z 1180.834,A 0.000,B 0.000,C 90.000,E1 6.087} C_DIS
LIN {X -0.187,Y -427.944,Z 1180.827,A 0.000,B 0.000,C 90.000,E1 4.878} C_DIS
LIN {X -0.136,Y -447.305,Z 1180.819,A 0.000,B 0.000,C 90.000,E1 3.440} C_DIS
LIN {X -0.109,Y -463.343,Z 1180.813,A 0.000,B 0.000,C 90.000,E1 2.293} C_DIS
LIN {X -0.060,Y -472.733,Z 1180.809,A 0.000,B 0.000,C 90.000,E1 1.604} C_DIS
LIN {X -0.210,Y -483.474,Z 1180.804,A 0.000,B 0.000,C 90.000,E1 0.802} C_DIS
LIN {X -0.025,Y -490.904,Z 1180.801,A 0.000,B 0.000,C 90.000,E1 0.172} C_DIS
LIN {X 0.107,Y -496.607,Z 1180.798,A 0.000,B 0.000,C 90.000,E1 359.656} C_DIS
LIN {X 0.001,Y -503.338,Z 1180.795,A 0.000,B 0.000,C 90.000,E1 359.026} C_DIS
LIN {X 0.199,Y -511.172,Z 1180.790,A 0.000,B 0.000,C 90.000,E1 358.167} C_DIS
LIN {X -0.138,Y -517.408,Z 1180.786,A 0.000,B 0.000,C 90.000,E1 357.478} C_DIS
LIN {X -0.272,Y -522.154,Z 1180.783,A 0.000,B 0.000,C 90.000,E1 356.906} C_DIS
LIN {X 0.141,Y -528.416,Z 1180.778,A 0.000,B 0.000,C 90.000,E1 355.988} C_DIS
LIN {X 0.119,Y -532.308,Z 1180.775,A 0.000,B 0.000,C 90.000,E1 355.412} C_DIS
LIN {X 0.129,Y -535.887,Z 1180.771,A 0.000,B 0.000,C 90.000,E1 354.837} C_DIS
LIN {X 0.163,Y -540.572,Z 1180.767,A 0.000,B 0.000,C 90.000,E1 353.976} C_DIS
LIN {X 0.293,Y -543.468,Z 1180.764,A 0.000,B 0.000,C 90.000,E1 353.394} C_DIS
LIN {X -0.155,Y -546.162,Z 1180.760,A 0.000,B 0.000,C 90.000,E1 352.875} C_DIS
LIN {X -0.208,Y -550.337,Z 1180.755,A 0.000,B 0.000,C 90.000,E1 351.894} C_DIS
LIN {X -0.077,Y -552.470,Z 1180.752,A 0.000,B 0.000,C 90.000,E1 351.319} C_DIS
LIN {X 0.277,Y -555.395,Z 1180.747,A 0.000,B 0.000,C 90.000,E1 350.443} C_DIS
LIN {X 0.024,Y -558.053,Z 1180.742,A 0.000,B 0.000,C 90.000,E1 349.634} C_DIS
LIN {X -0.103,Y -560.477,Z 1180.738,A 0.000,B 0.000,C 90.000,E1 348.814} C_DIS
LIN {X -0.046,Y -563.471,Z 1180.732,A 0.000,B 0.000,C 90.000,E1 347.701} C_DIS
LIN {X 0.052,Y -566.210,Z 1180.726,A 0.000,B 0.000,C 90.000,E1 346.589} C_DIS
LIN {X -0.056,Y -569.375,Z 1180.718,A 0.000,B 0.000,C 90.000,E1 345.227} C_DIS
LIN {X -0.110,Y -572.287,Z 1180.710,A 0.000,B 0.000,C 90.000,E1 343.866} C_DIS
LIN {X 0.042,Y -575.042,Z 1180.703,A 0.000,B 0.000,C 90.000,E1 342.489} C_DIS
LIN {X -0.124,Y -577.628,Z 1180.695,A 0.000,B 0.000,C 90.000,E1 341.148} C_DIS
LIN {X -0.077,Y -579.382,Z 1180.689,A 0.000,B 0.000,C 90.000,E1 340.061} C_DIS
LIN {X 0.192,Y -580.969,Z 1180.683,A 0.000,B 0.000,C 90.000,E1 338.954} C_DIS
LIN {X 0.087,Y -581.968,Z 1180.679,A 0.000,B 0.000,C 90.000,E1 338.156} C_DIS
LIN {X -0.011,Y -582.805,Z 1180.674,A 0.000,B 0.000,C 90.000,E1 337.358} C_DIS
LIN {X -0.241,Y -583.387,Z 1180.668,A 0.000,B 0.000,C 90.000,E1 336.305} C_DIS
LIN {X 0.030,Y -583.486,Z 1180.665,A 0.000,B 0.000,C 90.000,E1 335.741} C_DIS
LIN {X -0.227,Y -583.412,Z 1180.662,A 0.000,B 0.000,C 90.000,E1 335.229} C_DIS
LIN {X -0.084,Y -583.014,Z 1180.658,A 0.000,B 0.000,C 90.000,E1 334.409} C_DIS
LIN {X 0.183,Y -582.598,Z 1180.655,A 0.000,B 0.000,C 90.000,E1 333.845} C_DIS
LIN {X -0.078,Y -582.058,Z 1180.652,A 0.000,B 0.000,C 90.000,E1 333.332} C_DIS
LIN {X -0.208,Y -580.815,Z 1180.647,A 0.000,B 0.000,C 90.000,E1 332.538} C_DIS
LIN {X -0.103,Y -579.214,Z 1180.643,A 0.000,B 0.000,C 90.000,E1 331.719} C_DIS
LIN {X -0.254,Y -577.337,Z 1180.638,A 0.000,B 0.000,C 90.000,E1 330.923} C_DIS
LIN {X 0.080,Y -575.073,Z 1180.634,A 0.000,B 0.000,C 90.000,E1 330.078} C_DIS
LIN {X -0.111,Y -572.182,Z 1180.629,A 0.000,B 0.000,C 90.000,E1 329.282} C_DIS
LIN {X -0.071,Y -570.355,Z 1180.627,A 0.000,B 0.000,C 90.000,E1 328.869} C_DIS
LIN {X -0.033,Y -568.333,Z 1180.625,A 0.000,B 0.000,C 90.000,E1 328.456} C_DIS
LIN {X -0.202,Y -564.313,Z 1180.621,A 0.000,B 0.000,C 90.000,E1 327.788} C_DIS
LIN {X -0.301,Y -560.860,Z 1180.618,A 0.000,B 0.000,C 90.000,E1 327.248} C_DIS
LIN {X 0.310,Y -553.853,Z 1180.613,A 0.000,B 0.000,C 90.000,E1 326.215} C_DIS
LIN {X 0.005,Y -548.282,Z 1180.609,A 0.000,B 0.000,C 90.000,E1 325.548} C_DIS
LIN {X 0.058,Y -539.950,Z 1180.603,A 0.000,B 0.000,C 90.000,E1 324.562} C_DIS
LIN {X 0.093,Y -534.973,Z 1180.600,A 0.000,B 0.000,C 90.000,E1 323.989} C_DIS
LIN {X 0.158,Y -522.450,Z 1180.592,A 0.000,B 0.000,C 90.000,E1 322.557} C_DIS
LIN {X 0.231,Y -519.892,Z 1180.590,A 0.000,B 0.000,C 90.000,E1 322.190} C_DIS
LIN {X -0.123,Y -518.129,Z 1180.588,A 0.000,B 0.000,C 90.000,E1 321.904} C_DIS
LIN {X -0.180,Y -516.741,Z 1180.587,A 0.000,B 0.000,C 90.000,E1 321.618} C_DIS
LIN {X 0.270,Y -515.236,Z 1180.584,A 0.000,B 0.000,C 90.000,E1 321.090} C_DIS
LIN {X 0.054,Y -514.409,Z 1180.579,A 0.000,B 0.000,C 90.000,E1 320.231} C_DIS
LIN {X -0.238,Y -514.592,Z 1180.574,A 0.000,B 0.000,C 90.000,E1 319.380} C_DIS
LIN {X -0.137,Y -515.159,Z 1180.569,A 0.000,B 0.000,C 90.000,E1 318.485} C_DIS
LIN {X -0.069,Y -516.267,Z 1180.558,A 0.000,B 0.000,C 90.000,E1 316.419} C_DIS
LIN {X -0.240,Y -517.349,Z 1180.548,A 0.000,B 0.000,C 90.000,E1 314.676} C_DIS
LIN {X 0.062,Y -518.225,Z 1180.540,A 0.000,B 0.000,C 90.000,E1 313.176} C_DIS
LIN {X -0.139,Y -519.482,Z 1180.529,A 0.000,B 0.000,C 90.000,E1 311.148} C_DIS
LIN {X 0.135,Y -520.788,Z 1180.517,A 0.000,B 0.000,C 90.000,E1 309.072} C_DIS
LIN {X -0.150,Y -521.511,Z 1180.511,A 0.000,B 0.000,C 90.000,E1 307.935} C_DIS
LIN {X 0.033,Y -522.315,Z 1180.503,A 0.000,B 0.000,C 90.000,E1 306.457} C_DIS
LIN {X -0.186,Y -523.136,Z 1180.495,A 0.000,B 0.000,C 90.000,E1 305.025} C_DIS
LIN {X -0.267,Y -523.896,Z 1180.486,A 0.000,B 0.000,C 90.000,E1 303.579} C_DIS
LIN {X 0.111,Y -524.695,Z 1180.478,A 0.000,B 0.000,C 90.000,E1 302.084} C_DIS
LIN {X -0.221,Y -525.405,Z 1180.470,A 0.000,B 0.000,C 90.000,E1 300.669} C_DIS
LIN {X -0.095,Y -525.921,Z 1180.462,A 0.000,B 0.000,C 90.000,E1 299.205} C_DIS
LIN {X 0.089,Y -526.244,Z 1180.456,A 0.000,B 0.000,C 90.000,E1 298.025} C_DIS
LIN {X 0.031,Y -526.439,Z 1180.449,A 0.000,B 0.000,C 90.000,E1 296.873} C_DIS
LIN {X -0.161,Y -526.635,Z 1180.440,A 0.000,B 0.000,C 90.000,E1 295.155} C_DIS
LIN {X -0.048,Y -526.608,Z 1180.432,A 0.000,B 0.000,C 90.000,E1 293.695} C_DIS
LIN {X -0.008,Y -526.372,Z 1180.420,A 0.000,B 0.000,C 90.000,E1 291.663} C_DIS
LIN {X -0.143,Y -526.110,Z 1180.411,A 0.000,B 0.000,C 90.000,E1 289.939} C_DIS
LIN {X 0.028,Y -525.818,Z 1180.401,A 0.000,B 0.000,C 90.000,E1 288.181} C_DIS
LIN {X -0.138,Y -525.449,Z 1180.395,A 0.000,B 0.000,C 90.000,E1 287.040} C_DIS
LIN {X 0.192,Y -524.858,Z 1180.388,A 0.000,B 0.000,C 90.000,E1 285.843} C_DIS
LIN {X 0.008,Y -524.108,Z 1180.380,A 0.000,B 0.000,C 90.000,E1 284.411} C_DIS
LIN {X 0.052,Y -523.347,Z 1180.374,A 0.000,B 0.000,C 90.000,E1 283.244} C_DIS
LIN {X 0.237,Y -521.683,Z 1180.361,A 0.000,B 0.000,C 90.000,E1 280.894} C_DIS
LIN {X 0.171,Y -520.785,Z 1180.351,A 0.000,B 0.000,C 90.000,E1 279.151} C_DIS
LIN {X 0.078,Y -519.750,Z 1180.341,A 0.000,B 0.000,C 90.000,E1 277.409} C_DIS
LIN {X -0.175,Y -518.651,Z 1180.332,A 0.000,B 0.000,C 90.000,E1 275.682} C_DIS
LIN {X 0.066,Y -517.559,Z 1180.322,A 0.000,B 0.000,C 90.000,E1 273.898} C_DIS
LIN {X 0.151,Y -516.505,Z 1180.310,A 0.000,B 0.000,C 90.000,E1 271.835} C_DIS
LIN {X -0.165,Y -515.880,Z 1180.302,A 0.000,B 0.000,C 90.000,E1 270.401} C_DIS
LIN {X -0.132,Y -514.880,Z 1180.291,A 0.000,B 0.000,C 90.000,E1 268.339} C_DIS
LIN {X 0.107,Y -514.333,Z 1180.284,A 0.000,B 0.000,C 90.000,E1 267.135} C_DIS
LIN {X -0.221,Y -513.319,Z 1180.276,A 0.000,B 0.000,C 90.000,E1 265.698} C_DIS
LIN {X 0.077,Y -512.614,Z 1180.271,A 0.000,B 0.000,C 90.000,E1 264.780} C_DIS
LIN {X -0.230,Y -511.382,Z 1180.263,A 0.000,B 0.000,C 90.000,E1 263.337} C_DIS
LIN {X -0.011,Y -510.265,Z 1180.256,A 0.000,B 0.000,C 90.000,E1 262.129} C_DIS
LIN {X 0.167,Y -508.662,Z 1180.246,A 0.000,B 0.000,C 90.000,E1 260.330} C_DIS
LIN {X -0.192,Y -506.605,Z 1180.233,A 0.000,B 0.000,C 90.000,E1 257.993} C_DIS
LIN {X 0.157,Y -505.254,Z 1180.225,A 0.000,B 0.000,C 90.000,E1 256.464} C_DIS
LIN {X 0.043,Y -504.914,Z 1180.222,A 0.000,B 0.000,C 90.000,E1 255.880} C_DIS
LIN {X -0.079,Y -502.781,Z 1180.208,A 0.000,B 0.000,C 90.000,E1 253.504} C_DIS
LIN {X -0.013,Y -501.997,Z 1180.203,A 0.000,B 0.000,C 90.000,E1 252.598} C_DIS
LIN {X -0.024,Y -501.632,Z 1180.200,A 0.000,B 0.000,C 90.000,E1 252.000} C_DIS
LIN {X 0.144,Y -499.818,Z 1180.188,A 0.000,B 0.000,C 90.000,E1 249.880} C_DIS
LIN {X -0.230,Y -498.648,Z 1180.182,A 0.000,B 0.000,C 90.000,E1 248.720} C_DIS
LIN {X 0.140,Y -496.874,Z 1180.172,A 0.000,B 0.000,C 90.000,E1 246.869} C_DIS
LIN {X 0.105,Y -495.686,Z 1180.165,A 0.000,B 0.000,C 90.000,E1 245.665} C_DIS
LIN {X 0.142,Y -493.607,Z 1180.155,A 0.000,B 0.000,C 90.000,E1 243.845} C_DIS
LIN {X -0.158,Y -492.053,Z 1180.148,A 0.000,B 0.000,C 90.000,E1 242.666} C_DIS
LIN {X -0.192,Y -489.297,Z 1180.136,A 0.000,B 0.000,C 90.000,E1 240.539} C_DIS
LIN {X 0.178,Y -486.790,Z 1180.126,A 0.000,B 0.000,C 90.000,E1 238.663} C_DIS
LIN {X -0.146,Y -484.653,Z 1180.118,A 0.000,B 0.000,C 90.000,E1 237.168} C_DIS
LIN {X 0.000,Y -481.262,Z 1180.104,A 0.000,B 0.000,C 90.000,E1 234.689} C_DIS
LIN {X 0.115,Y -479.185,Z 1180.095,A 0.000,B 0.000,C 90.000,E1 233.130} C_DIS
LIN {X 0.164,Y -475.776,Z 1180.082,A 0.000,B 0.000,C 90.000,E1 230.642} C_DIS
LIN {X 0.083,Y -473.843,Z 1180.073,A 0.000,B 0.000,C 90.000,E1 229.094} C_DIS
LIN {X 0.140,Y -472.098,Z 1180.066,A 0.000,B 0.000,C 90.000,E1 227.838} C_DIS
LIN {X -0.246,Y -467.279,Z 1180.047,A 0.000,B 0.000,C 90.000,E1 224.433} C_DIS
LIN {X 0.066,Y -464.421,Z 1180.031,A 0.000,B 0.000,C 90.000,E1 221.553} C_DIS
LIN {X -0.274,Y -462.771,Z 1180.006,A 0.000,B 0.000,C 90.000,E1 217.156} C_DIS
LIN {X -0.089,Y -463.062,Z 1179.978,A 0.000,B 0.000,C 90.000,E1 212.054} C_DIS
LIN {X 0.095,Y -464.297,Z 1179.968,A 0.000,B 0.000,C 90.000,E1 210.129} C_DIS
LIN {X 0.228,Y -466.173,Z 1179.955,A 0.000,B 0.000,C 90.000,E1 207.897} C_DIS
LIN {X -0.027,Y -471.836,Z 1179.929,A 0.000,B 0.000,C 90.000,E1 203.206} C_DIS
LIN {X 0.076,Y -478.810,Z 1179.908,A 0.000,B 0.000,C 90.000,E1 199.450} C_DIS
LIN {X -0.127,Y -487.354,Z 1179.889,A 0.000,B 0.000,C 90.000,E1 196.079} C_DIS
LIN {X 0.177,Y -495.657,Z 1179.874,A 0.000,B 0.000,C 90.000,E1 193.300} C_DIS
LIN {X -0.224,Y -501.476,Z 1179.864,A 0.000,B 0.000,C 90.000,E1 191.535} C_DIS
LIN {X 0.001,Y -505.453,Z 1179.857,A 0.000,B 0.000,C 90.000,E1 190.310} C_DIS
LIN {X 0.080,Y -512.626,Z 1179.846,A 0.000,B 0.000,C 90.000,E1 188.219} C_DIS
LIN {X -0.207,Y -517.804,Z 1179.838,A 0.000,B 0.000,C 90.000,E1 186.777} C_DIS
LIN {X 0.059,Y -523.799,Z 1179.828,A 0.000,B 0.000,C 90.000,E1 184.992} C_DIS
LIN {X -0.103,Y -529.838,Z 1179.818,A 0.000,B 0.000,C 90.000,E1 183.269} C_DIS
LIN {X -0.157,Y -534.862,Z 1179.810,A 0.000,B 0.000,C 90.000,E1 181.835} C_DIS
LIN {X -0.110,Y -540.785,Z 1179.801,A 0.000,B 0.000,C 90.000,E1 180.115} C_DIS
LIN {X -0.043,Y -543.823,Z 1179.796,A 0.000,B 0.000,C 90.000,E1 179.255} C_DIS
LIN {X 0.155,Y -548.784,Z 1179.788,A 0.000,B 0.000,C 90.000,E1 177.822} C_DIS
LIN {X -0.164,Y -552.701,Z 1179.782,A 0.000,B 0.000,C 90.000,E1 176.731} C_DIS
LIN {X -0.248,Y -558.518,Z 1179.772,A 0.000,B 0.000,C 90.000,E1 175.065} C_DIS
LIN {X -0.160,Y -564.271,Z 1179.763,A 0.000,B 0.000,C 90.000,E1 173.394} C_DIS
LIN {X 0.041,Y -569.920,Z 1179.754,A 0.000,B 0.000,C 90.000,E1 171.724} C_DIS
LIN {X -0.242,Y -574.653,Z 1179.746,A 0.000,B 0.000,C 90.000,E1 170.387} C_DIS
LIN {X 0.125,Y -579.212,Z 1179.739,A 0.000,B 0.000,C 90.000,E1 168.993} C_DIS
LIN {X 0.115,Y -583.749,Z 1179.731,A 0.000,B 0.000,C 90.000,E1 167.645} C_DIS
LIN {X 0.184,Y -588.288,Z 1179.724,A 0.000,B 0.000,C 90.000,E1 166.297} C_DIS
LIN {X -0.102,Y -592.654,Z 1179.717,A 0.000,B 0.000,C 90.000,E1 164.991} C_DIS
LIN {X 0.132,Y -597.863,Z 1179.708,A 0.000,B 0.000,C 90.000,E1 163.378} C_DIS
LIN {X -0.097,Y -602.950,Z 1179.699,A 0.000,B 0.000,C 90.000,E1 161.819} C_DIS
LIN {X -0.037,Y -607.815,Z 1179.690,A 0.000,B 0.000,C 90.000,E1 160.242} C_DIS
LIN {X -0.186,Y -611.752,Z 1179.683,A 0.000,B 0.000,C 90.000,E1 158.954} C_DIS
LIN {X 0.265,Y -616.332,Z 1179.674,A 0.000,B 0.000,C 90.000,E1 157.358} C_DIS
LIN {X -0.047,Y -618.642,Z 1179.670,A 0.000,B 0.000,C 90.000,E1 156.613} C_DIS
LIN {X 0.207,Y -623.069,Z 1179.661,A 0.000,B 0.000,C 90.000,E1 155.049} C_DIS
LIN {X 0.269,Y -627.878,Z 1179.652,A 0.000,B 0.000,C 90.000,E1 153.256} C_DIS
LIN {X -0.227,Y -629.940,Z 1179.647,A 0.000,B 0.000,C 90.000,E1 152.538} C_DIS
LIN {X -0.081,Y -633.291,Z 1179.640,A 0.000,B 0.000,C 90.000,E1 151.257} C_DIS
LIN {X -0.176,Y -635.812,Z 1179.635,A 0.000,B 0.000,C 90.000,E1 150.255} C_DIS
LIN {X 0.319,Y -638.278,Z 1179.629,A 0.000,B 0.000,C 90.000,E1 149.203} C_DIS
LIN {X -0.150,Y -641.652,Z 1179.621,A 0.000,B 0.000,C 90.000,E1 147.740} C_DIS
LIN {X -0.276,Y -644.230,Z 1179.614,A 0.000,B 0.000,C 90.000,E1 146.501} C_DIS
LIN {X 0.064,Y -647.117,Z 1179.605,A 0.000,B 0.000,C 90.000,E1 144.975} C_DIS
LIN {X -0.071,Y -649.822,Z 1179.597,A 0.000,B 0.000,C 90.000,E1 143.497} C_DIS
LIN {X 0.234,Y -652.426,Z 1179.589,A 0.000,B 0.000,C 90.000,E1 141.984} C_DIS
LIN {X 0.091,Y -654.234,Z 1179.583,A 0.000,B 0.000,C 90.000,E1 141.009} C_DIS
LIN {X -0.106,Y -658.059,Z 1179.573,A 0.000,B 0.000,C 90.000,E1 139.057} C_DIS
LIN {X 0.249,Y -661.737,Z 1179.563,A 0.000,B 0.000,C 90.000,E1 137.310} C_DIS
LIN {X -0.287,Y -664.777,Z 1179.555,A 0.000,B 0.000,C 90.000,E1 135.891} C_DIS
LIN {X -0.289,Y -669.580,Z 1179.543,A 0.000,B 0.000,C 90.000,E1 133.704} C_DIS
LIN {X -0.150,Y -674.191,Z 1179.532,A 0.000,B 0.000,C 90.000,E1 131.757} C_DIS
LIN {X 0.201,Y -679.359,Z 1179.520,A 0.000,B 0.000,C 90.000,E1 129.564} C_DIS
LIN {X -0.377,Y -682.946,Z 1179.512,A 0.000,B 0.000,C 90.000,E1 128.177} C_DIS
LIN {X -0.310,Y -687.140,Z 1179.503,A 0.000,B 0.000,C 90.000,E1 126.503} C_DIS
LIN {X 0.356,Y -690.663,Z 1179.495,A 0.000,B 0.000,C 90.000,E1 125.025} C_DIS
LIN {X -0.124,Y -692.918,Z 1179.490,A 0.000,B 0.000,C 90.000,E1 124.119} C_DIS
LIN {X 0.262,Y -696.042,Z 1179.482,A 0.000,B 0.000,C 90.000,E1 122.673} C_DIS
LIN {X 0.056,Y -698.053,Z 1179.476,A 0.000,B 0.000,C 90.000,E1 121.750} C_DIS
LIN {X -0.094,Y -700.400,Z 1179.470,A 0.000,B 0.000,C 90.000,E1 120.590} C_DIS
LIN {X -0.238,Y -702.009,Z 1179.465,A 0.000,B 0.000,C 90.000,E1 119.667} C_DIS
LIN {X -0.083,Y -703.930,Z 1179.458,A 0.000,B 0.000,C 90.000,E1 118.487} C_DIS
LIN {X 0.435,Y -705.349,Z 1179.453,A 0.000,B 0.000,C 90.000,E1 117.513} C_DIS
LIN {X -0.272,Y -706.105,Z 1179.449,A 0.000,B 0.000,C 90.000,E1 116.873} C_DIS
LIN {X -0.043,Y -706.599,Z 1179.444,A 0.000,B 0.000,C 90.000,E1 115.924} C_DIS
LIN {X -0.091,Y -706.700,Z 1179.442,A 0.000,B 0.000,C 90.000,E1 115.463} C_DIS
LIN {X 0.198,Y -706.653,Z 1179.439,A 0.000,B 0.000,C 90.000,E1 114.975} C_DIS
LIN {X 0.144,Y -706.379,Z 1179.436,A 0.000,B 0.000,C 90.000,E1 114.515} C_DIS
LIN {X -0.207,Y -705.515,Z 1179.434,A 0.000,B 0.000,C 90.000,E1 114.079} C_DIS
LIN {X 0.082,Y -704.881,Z 1179.432,A 0.000,B 0.000,C 90.000,E1 113.823} C_DIS
LIN {X -0.276,Y -702.855,Z 1179.430,A 0.000,B 0.000,C 90.000,E1 113.387} C_DIS
LIN {X -0.137,Y -702.192,Z 1179.429,A 0.000,B 0.000,C 90.000,E1 113.259} C_DIS
LIN {X 0.002,Y -701.195,Z 1179.429,A 0.000,B 0.000,C 90.000,E1 113.131} C_DIS
LIN {X 0.341,Y -696.171,Z 1179.426,A 0.000,B 0.000,C 90.000,E1 112.642} C_DIS
LIN {X -0.360,Y -694.353,Z 1179.425,A 0.000,B 0.000,C 90.000,E1 112.589} C_DIS
LIN {X 0.055,Y -689.165,Z 1179.424,A 0.000,B 0.000,C 90.000,E1 112.386} C_DIS
LIN {X 0.028,Y -685.433,Z 1179.424,A 0.000,B 0.000,C 90.000,E1 112.280} C_DIS
LIN {X -0.209,Y -683.974,Z 1179.424,A 0.000,B 0.000,C 90.000,E1 112.280} C_DIS
LIN {X 0.365,Y -677.574,Z 1179.424,A 0.000,B 0.000,C 90.000,E1 112.206} C_DIS
LIN {X 0.283,Y -605.739,Z 1179.424,A 0.000,B 0.000,C 90.000,E1 112.206} C_DIS
LIN {X 0.344,Y -601.212,Z 1179.422,A 0.000,B 0.000,C 90.000,E1 111.897} C_DIS
LIN {X 0.286,Y -583.791,Z 1179.414,A 0.000,B 0.000,C 90.000,E1 110.482} C_DIS
LIN {X 0.255,Y -575.450,Z 1179.410,A 0.000,B 0.000,C 90.000,E1 109.812} C_DIS
LIN {X -0.354,Y -566.299,Z 1179.407,A 0.000,B 0.000,C 90.000,E1 109.214} C_DIS
LIN {X -0.036,Y -557.351,Z 1179.403,A 0.000,B 0.000,C 90.000,E1 108.544} C_DIS
LIN {X 0.101,Y -552.728,Z 1179.401,A 0.000,B 0.000,C 90.000,E1 108.127} C_DIS
LIN {X -0.073,Y -551.341,Z 1179.399,A 0.000,B 0.000,C 90.000,E1 107.873} C_DIS
LIN {X -0.147,Y -550.519,Z 1179.397,A 0.000,B 0.000,C 90.000,E1 107.457} C_DIS
LIN {X 0.213,Y -550.525,Z 1179.394,A 0.000,B 0.000,C 90.000,E1 106.858} C_DIS
LIN {X 0.030,Y -552.713,Z 1179.380,A 0.000,B 0.000,C 90.000,E1 104.356} C_DIS
LIN {X -0.202,Y -554.121,Z 1179.370,A 0.000,B 0.000,C 90.000,E1 102.703} C_DIS
LIN {X -0.239,Y -556.707,Z 1179.357,A 0.000,B 0.000,C 90.000,E1 100.197} C_DIS
LIN {X -0.062,Y -558.401,Z 1179.347,A 0.000,B 0.000,C 90.000,E1 98.511} C_DIS
LIN {X -0.142,Y -559.429,Z 1179.341,A 0.000,B 0.000,C 90.000,E1 97.409} C_DIS
LIN {X -0.145,Y -560.568,Z 1179.333,A 0.000,B 0.000,C 90.000,E1 96.024} C_DIS
LIN {X -0.004,Y -561.865,Z 1179.323,A 0.000,B 0.000,C 90.000,E1 94.073} C_DIS
LIN {X -0.276,Y -563.454,Z 1179.310,A 0.000,B 0.000,C 90.000,E1 91.892} C_DIS
LIN {X 0.270,Y -564.495,Z 1179.303,A 0.000,B 0.000,C 90.000,E1 90.458} C_DIS
LIN {X -0.196,Y -565.671,Z 1179.294,A 0.000,B 0.000,C 90.000,E1 88.854} C_DIS
LIN {X 0.275,Y -566.379,Z 1179.287,A 0.000,B 0.000,C 90.000,E1 87.707} C_DIS
LIN {X 0.196,Y -567.134,Z 1179.281,A 0.000,B 0.000,C 90.000,E1 86.617} C_DIS
LIN {X 0.236,Y -568.048,Z 1179.274,A 0.000,B 0.000,C 90.000,E1 85.241} C_DIS
LIN {X -0.180,Y -569.001,Z 1179.266,A 0.000,B 0.000,C 90.000,E1 83.913} C_DIS
LIN {X 0.105,Y -570.159,Z 1179.257,A 0.000,B 0.000,C 90.000,E1 82.243} C_DIS
LIN {X -0.184,Y -570.995,Z 1179.249,A 0.000,B 0.000,C 90.000,E1 80.905} C_DIS
LIN {X -0.171,Y -572.042,Z 1179.239,A 0.000,B 0.000,C 90.000,E1 78.993} C_DIS
LIN {X -0.124,Y -572.857,Z 1179.230,A 0.000,B 0.000,C 90.000,E1 77.353} C_DIS
LIN {X 0.074,Y -573.741,Z 1179.221,A 0.000,B 0.000,C 90.000,E1 75.700} C_DIS
LIN {X -0.104,Y -574.315,Z 1179.215,A 0.000,B 0.000,C 90.000,E1 74.629} C_DIS
LIN {X -0.078,Y -575.597,Z 1179.201,A 0.000,B 0.000,C 90.000,E1 72.181} C_DIS
LIN {X -0.051,Y -576.581,Z 1179.192,A 0.000,B 0.000,C 90.000,E1 70.550} C_DIS
LIN {X 0.175,Y -577.363,Z 1179.186,A 0.000,B 0.000,C 90.000,E1 69.444} C_DIS
LIN {X 0.006,Y -580.081,Z 1179.169,A 0.000,B 0.000,C 90.000,E1 66.485} C_DIS
LIN {X 0.114,Y -580.878,Z 1179.165,A 0.000,B 0.000,C 90.000,E1 65.665} C_DIS
LIN {X 0.228,Y -582.611,Z 1179.154,A 0.000,B 0.000,C 90.000,E1 63.768} C_DIS
LIN {X 0.100,Y -583.914,Z 1179.147,A 0.000,B 0.000,C 90.000,E1 62.436} C_DIS
LIN {X -0.099,Y -585.488,Z 1179.138,A 0.000,B 0.000,C 90.000,E1 60.845} C_DIS
LIN {X 0.080,Y -586.628,Z 1179.131,A 0.000,B 0.000,C 90.000,E1 59.488} C_DIS
LIN {X 0.059,Y -587.757,Z 1179.123,A 0.000,B 0.000,C 90.000,E1 58.152} C_DIS
LIN {X 0.070,Y -588.865,Z 1179.114,A 0.000,B 0.000,C 90.000,E1 56.548} C_DIS
LIN {X 0.206,Y -589.613,Z 1179.108,A 0.000,B 0.000,C 90.000,E1 55.468} C_DIS
LIN {X 0.199,Y -590.372,Z 1179.102,A 0.000,B 0.000,C 90.000,E1 54.402} C_DIS
LIN {X 0.060,Y -591.273,Z 1179.095,A 0.000,B 0.000,C 90.000,E1 53.084} C_DIS
LIN {X -0.018,Y -592.583,Z 1179.083,A 0.000,B 0.000,C 90.000,E1 50.964} C_DIS
LIN {X 0.129,Y -593.228,Z 1179.076,A 0.000,B 0.000,C 90.000,E1 49.622} C_DIS
LIN {X -0.162,Y -593.722,Z 1179.068,A 0.000,B 0.000,C 90.000,E1 48.324} C_DIS
LIN {X -0.043,Y -593.994,Z 1179.061,A 0.000,B 0.000,C 90.000,E1 46.986} C_DIS
LIN {X -0.300,Y -594.046,Z 1179.057,A 0.000,B 0.000,C 90.000,E1 46.215} C_DIS
LIN {X 0.238,Y -593.906,Z 1179.049,A 0.000,B 0.000,C 90.000,E1 44.838} C_DIS
LIN {X 0.161,Y -593.643,Z 1179.043,A 0.000,B 0.000,C 90.000,E1 43.785} C_DIS
LIN {X -0.332,Y -593.070,Z 1179.037,A 0.000,B 0.000,C 90.000,E1 42.771} C_DIS
LIN {X 0.213,Y -592.200,Z 1179.030,A 0.000,B 0.000,C 90.000,E1 41.391} C_DIS
LIN {X -0.060,Y -591.602,Z 1179.026,A 0.000,B 0.000,C 90.000,E1 40.620} C_DIS
LIN {X 0.068,Y -590.302,Z 1179.018,A 0.000,B 0.000,C 90.000,E1 39.277} C_DIS
LIN {X -0.035,Y -589.067,Z 1179.012,A 0.000,B 0.000,C 90.000,E1 38.222} C_DIS
LIN {X -0.256,Y -588.035,Z 1179.008,A 0.000,B 0.000,C 90.000,E1 37.443} C_DIS
LIN {X -0.287,Y -586.326,Z 1179.002,A 0.000,B 0.000,C 90.000,E1 36.377} C_DIS
LIN {X -0.342,Y -584.334,Z 1178.996,A 0.000,B 0.000,C 90.000,E1 35.311} C_DIS
LIN {X -0.126,Y -582.515,Z 1178.992,A 0.000,B 0.000,C 90.000,E1 34.485} C_DIS
LIN {X 0.073,Y -580.442,Z 1178.987,A 0.000,B 0.000,C 90.000,E1 33.658} C_DIS
LIN {X 0.087,Y -578.849,Z 1178.984,A 0.000,B 0.000,C 90.000,E1 33.118} C_DIS
LIN {X -0.242,Y -576.181,Z 1178.980,A 0.000,B 0.000,C 90.000,E1 32.339} C_DIS
LIN {X -0.257,Y -574.241,Z 1178.977,A 0.000,B 0.000,C 90.000,E1 31.799} C_DIS
LIN {X 0.204,Y -572.118,Z 1178.974,A 0.000,B 0.000,C 90.000,E1 31.209} C_DIS
LIN {X 0.073,Y -569.142,Z 1178.970,A 0.000,B 0.000,C 90.000,E1 30.541} C_DIS
LIN {X 0.010,Y -564.567,Z 1178.964,A 0.000,B 0.000,C 90.000,E1 29.589} C_DIS
LIN {X 0.092,Y -559.277,Z 1178.959,A 0.000,B 0.000,C 90.000,E1 28.615} C_DIS
LIN {X 0.220,Y -554.404,Z 1178.954,A 0.000,B 0.000,C 90.000,E1 27.769} C_DIS
LIN {X -0.221,Y -550.937,Z 1178.951,A 0.000,B 0.000,C 90.000,E1 27.257} C_DIS
LIN {X 0.056,Y -547.118,Z 1178.948,A 0.000,B 0.000,C 90.000,E1 26.668} C_DIS
LIN {X -0.067,Y -541.994,Z 1178.944,A 0.000,B 0.000,C 90.000,E1 25.976} C_DIS
LIN {X -0.097,Y -537.694,Z 1178.941,A 0.000,B 0.000,C 90.000,E1 25.412} C_DIS
LIN {X 0.210,Y -534.264,Z 1178.939,A 0.000,B 0.000,C 90.000,E1 24.951} C_DIS
LIN {X 0.215,Y -525.691,Z 1178.933,A 0.000,B 0.000,C 90.000,E1 23.951} C_DIS
LIN {X 0.121,Y -520.596,Z 1178.930,A 0.000,B 0.000,C 90.000,E1 23.387} C_DIS
LIN {X 0.075,Y -513.982,Z 1178.926,A 0.000,B 0.000,C 90.000,E1 22.695} C_DIS
LIN {X -0.188,Y -505.887,Z 1178.922,A 0.000,B 0.000,C 90.000,E1 21.897} C_DIS
LIN {X -0.247,Y -497.663,Z 1178.917,A 0.000,B 0.000,C 90.000,E1 21.099} C_DIS
LIN {X 0.246,Y -487.722,Z 1178.912,A 0.000,B 0.000,C 90.000,E1 20.120} C_DIS
LIN {X 0.058,Y -477.411,Z 1178.907,A 0.000,B 0.000,C 90.000,E1 19.214} C_DIS
LIN {X -0.097,Y -470.335,Z 1178.903,A 0.000,B 0.000,C 90.000,E1 18.598} C_DIS
LIN {X 0.017,Y -451.765,Z 1178.894,A 0.000,B 0.000,C 90.000,E1 16.913} C_DIS
LIN {X -0.072,Y -428.623,Z 1178.881,A 0.000,B 0.000,C 90.000,E1 14.662} C_DIS
LIN {X 0.151,Y -414.927,Z 1178.873,A 0.000,B 0.000,C 90.000,E1 13.119} C_DIS
LIN {X -0.028,Y -402.994,Z 1178.865,A 0.000,B 0.000,C 90.000,E1 11.658} C_DIS
LIN {X 0.000,Y -396.881,Z 1178.860,A 0.000,B 0.000,C 90.000,E1 10.782} C_DIS
LIN {X 0.003,Y -394.089,Z 1178.857,A 0.000,B 0.000,C 90.000,E1 10.254} C_DIS
LIN {X -0.163,Y -393.008,Z 1178.855,A 0.000,B 0.000,C 90.000,E1 9.905} C_DIS
LIN {X -0.201,Y -393.002,Z 1178.855,A 0.000,B 0.000,C 90.000,E1 9.905} C_DIS
LIN {X -0.013,Y -393.238,Z 1178.853,A 0.000,B 0.000,C 90.000,E1 9.557} C_DIS
LIN {X 0.000,Y -393.498,Z 1178.852,A 0.000,B 0.000,C 90.000,E1 9.378} C_DIS
LIN {X 0.107,Y -394.790,Z 1178.849,A 0.000,B 0.000,C 90.000,E1 8.803} C_DIS
LIN {X -0.003,Y -398.159,Z 1178.844,A 0.000,B 0.000,C 90.000,E1 7.936} C_DIS
LIN {X -0.079,Y -402.520,Z 1178.839,A 0.000,B 0.000,C 90.000,E1 7.068} C_DIS
LIN {X -0.145,Y -406.599,Z 1178.836,A 0.000,B 0.000,C 90.000,E1 6.543} C_DIS
LIN {X -0.038,Y -413.028,Z 1178.833,A 0.000,B 0.000,C 90.000,E1 5.967} C_DIS
LIN {X 0.008,Y -430.192,Z 1178.826,A 0.000,B 0.000,C 90.000,E1 4.645} C_DIS
LIN {X 0.212,Y -449.306,Z 1178.818,A 0.000,B 0.000,C 90.000,E1 3.212} C_DIS
LIN {X -0.211,Y -462.220,Z 1178.813,A 0.000,B 0.000,C 90.000,E1 2.350} C_DIS
LIN {X -0.190,Y -471.728,Z 1178.809,A 0.000,B 0.000,C 90.000,E1 1.661} C_DIS
LIN {X -0.225,Y -482.409,Z 1178.805,A 0.000,B 0.000,C 90.000,E1 0.859} C_DIS
LIN {X -0.016,Y -489.971,Z 1178.801,A 0.000,B 0.000,C 90.000,E1 0.229} C_DIS
LIN {X 0.078,Y -496.440,Z 1178.798,A 0.000,B 0.000,C 90.000,E1 359.656} C_DIS
LIN {X -0.208,Y -503.477,Z 1178.795,A 0.000,B 0.000,C 90.000,E1 359.026} C_DIS
LIN {X 0.047,Y -511.303,Z 1178.790,A 0.000,B 0.000,C 90.000,E1 358.165} C_DIS
LIN {X 0.212,Y -517.591,Z 1178.786,A 0.000,B 0.000,C 90.000,E1 357.421} C_DIS
LIN {X 0.121,Y -522.357,Z 1178.783,A 0.000,B 0.000,C 90.000,E1 356.846} C_DIS
LIN {X -0.016,Y -528.632,Z 1178.778,A 0.000,B 0.000,C 90.000,E1 355.988} C_DIS
LIN {X -0.037,Y -532.548,Z 1178.775,A 0.000,B 0.000,C 90.000,E1 355.412} C_DIS
LIN {X -0.027,Y -536.147,Z 1178.771,A 0.000,B 0.000,C 90.000,E1 354.837} C_DIS
LIN {X -0.259,Y -540.155,Z 1178.767,A 0.000,B 0.000,C 90.000,E1 354.147} C_DIS
LIN {X 0.142,Y -543.774,Z 1178.763,A 0.000,B 0.000,C 90.000,E1 353.394} C_DIS
LIN {X 0.237,Y -546.479,Z 1178.760,A 0.000,B 0.000,C 90.000,E1 352.818} C_DIS
LIN {X 0.088,Y -549.505,Z 1178.756,A 0.000,B 0.000,C 90.000,E1 352.129} C_DIS
LIN {X -0.250,Y -551.806,Z 1178.753,A 0.000,B 0.000,C 90.000,E1 351.602} C_DIS
LIN {X 0.010,Y -554.801,Z 1178.749,A 0.000,B 0.000,C 90.000,E1 350.735} C_DIS
LIN {X -0.250,Y -557.555,Z 1178.744,A 0.000,B 0.000,C 90.000,E1 349.926} C_DIS
LIN {X 0.164,Y -560.073,Z 1178.739,A 0.000,B 0.000,C 90.000,E1 349.050} C_DIS
LIN {X 0.216,Y -563.134,Z 1178.733,A 0.000,B 0.000,C 90.000,E1 347.937} C_DIS
LIN {X -0.241,Y -565.935,Z 1178.727,A 0.000,B 0.000,C 90.000,E1 346.881} C_DIS
LIN {X -0.176,Y -569.784,Z 1178.718,A 0.000,B 0.000,C 90.000,E1 345.227} C_DIS
LIN {X 0.143,Y -572.152,Z 1178.712,A 0.000,B 0.000,C 90.000,E1 344.102} C_DIS
LIN {X -0.253,Y -574.939,Z 1178.704,A 0.000,B 0.000,C 90.000,E1 342.779} C_DIS
LIN {X -0.052,Y -577.585,Z 1178.697,A 0.000,B 0.000,C 90.000,E1 341.402} C_DIS
LIN {X -0.011,Y -579.436,Z 1178.691,A 0.000,B 0.000,C 90.000,E1 340.315} C_DIS
LIN {X 0.253,Y -581.108,Z 1178.685,A 0.000,B 0.000,C 90.000,E1 339.209} C_DIS
LIN {X 0.147,Y -582.152,Z 1178.680,A 0.000,B 0.000,C 90.000,E1 338.411} C_DIS
LIN {X 0.048,Y -583.082,Z 1178.676,A 0.000,B 0.000,C 90.000,E1 337.614} C_DIS
LIN {X 0.183,Y -583.675,Z 1178.671,A 0.000,B 0.000,C 90.000,E1 336.794} C_DIS
LIN {X 0.093,Y -584.040,Z 1178.667,A 0.000,B 0.000,C 90.000,E1 335.997} C_DIS
LIN {X -0.163,Y -584.094,Z 1178.664,A 0.000,B 0.000,C 90.000,E1 335.485} C_DIS
LIN {X -0.139,Y -583.643,Z 1178.658,A 0.000,B 0.000,C 90.000,E1 334.409} C_DIS
LIN {X 0.004,Y -582.992,Z 1178.653,A 0.000,B 0.000,C 90.000,E1 333.589} C_DIS
LIN {X 0.010,Y -582.336,Z 1178.650,A 0.000,B 0.000,C 90.000,E1 333.050} C_DIS
LIN {X 0.136,Y -581.036,Z 1178.646,A 0.000,B 0.000,C 90.000,E1 332.231} C_DIS
LIN {X 0.003,Y -579.360,Z 1178.641,A 0.000,B 0.000,C 90.000,E1 331.435} C_DIS
LIN {X -0.278,Y -578.108,Z 1178.638,A 0.000,B 0.000,C 90.000,E1 330.923} C_DIS
LIN {X 0.065,Y -575.887,Z 1178.634,A 0.000,B 0.000,C 90.000,E1 330.078} C_DIS
LIN {X 0.042,Y -574.008,Z 1178.631,A 0.000,B 0.000,C 90.000,E1 329.537} C_DIS
LIN {X -0.119,Y -573.040,Z 1178.629,A 0.000,B 0.000,C 90.000,E1 329.282} C_DIS
LIN {X -0.157,Y -570.581,Z 1178.626,A 0.000,B 0.000,C 90.000,E1 328.742} C_DIS
LIN {X -0.126,Y -568.427,Z 1178.624,A 0.000,B 0.000,C 90.000,E1 328.329} C_DIS
LIN {X -0.292,Y -564.472,Z 1178.620,A 0.000,B 0.000,C 90.000,E1 327.661} C_DIS
LIN {X -0.087,Y -560.885,Z 1178.617,A 0.000,B 0.000,C 90.000,E1 327.089} C_DIS
LIN {X -0.243,Y -555.087,Z 1178.613,A 0.000,B 0.000,C 90.000,E1 326.294} C_DIS
LIN {X -0.289,Y -551.840,Z 1178.610,A 0.000,B 0.000,C 90.000,E1 325.881} C_DIS
LIN {X -0.295,Y -546.071,Z 1178.606,A 0.000,B 0.000,C 90.000,E1 325.182} C_DIS
LIN {X -0.271,Y -537.591,Z 1178.601,A 0.000,B 0.000,C 90.000,E1 324.196} C_DIS
LIN {X -0.156,Y -523.891,Z 1178.592,A 0.000,B 0.000,C 90.000,E1 322.637} C_DIS
LIN {X -0.051,Y -520.668,Z 1178.590,A 0.000,B 0.000,C 90.000,E1 322.190} C_DIS
LIN {X 0.087,Y -519.748,Z 1178.589,A 0.000,B 0.000,C 90.000,E1 322.029} C_DIS
LIN {X 0.228,Y -517.285,Z 1178.587,A 0.000,B 0.000,C 90.000,E1 321.537} C_DIS
LIN {X 0.164,Y -515.853,Z 1178.584,A 0.000,B 0.000,C 90.000,E1 321.090} C_DIS
LIN {X 0.098,Y -515.409,Z 1178.582,A 0.000,B 0.000,C 90.000,E1 320.803} C_DIS
LIN {X -0.047,Y -514.811,Z 1178.579,A 0.000,B 0.000,C 90.000,E1 320.231} C_DIS
LIN {X 0.057,Y -514.957,Z 1178.574,A 0.000,B 0.000,C 90.000,E1 319.337} C_DIS
LIN {X 0.035,Y -515.659,Z 1178.568,A 0.000,B 0.000,C 90.000,E1 318.162} C_DIS
LIN {X 0.038,Y -516.959,Z 1178.555,A 0.000,B 0.000,C 90.000,E1 315.810} C_DIS
LIN {X -0.038,Y -517.865,Z 1178.546,A 0.000,B 0.000,C 90.000,E1 314.352} C_DIS
LIN {X 0.274,Y -518.702,Z 1178.538,A 0.000,B 0.000,C 90.000,E1 312.852} C_DIS
LIN {X -0.201,Y -519.807,Z 1178.529,A 0.000,B 0.000,C 90.000,E1 311.148} C_DIS
LIN {X 0.081,Y -521.084,Z 1178.517,A 0.000,B 0.000,C 90.000,E1 309.072} C_DIS
LIN {X 0.166,Y -522.001,Z 1178.509,A 0.000,B 0.000,C 90.000,E1 307.604} C_DIS
LIN {X -0.097,Y -522.983,Z 1178.499,A 0.000,B 0.000,C 90.000,E1 305.884} C_DIS
LIN {X 0.035,Y -524.097,Z 1178.488,A 0.000,B 0.000,C 90.000,E1 303.833} C_DIS
LIN {X 0.085,Y -525.041,Z 1178.478,A 0.000,B 0.000,C 90.000,E1 302.084} C_DIS
LIN {X -0.242,Y -525.776,Z 1178.470,A 0.000,B 0.000,C 90.000,E1 300.669} C_DIS
LIN {X 0.204,Y -526.211,Z 1178.464,A 0.000,B 0.000,C 90.000,E1 299.461} C_DIS
LIN {X 0.081,Y -526.644,Z 1178.456,A 0.000,B 0.000,C 90.000,E1 298.025} C_DIS
LIN {X -0.277,Y -526.873,Z 1178.448,A 0.000,B 0.000,C 90.000,E1 296.616} C_DIS
LIN {X -0.155,Y -527.046,Z 1178.440,A 0.000,B 0.000,C 90.000,E1 295.155} C_DIS
LIN {X -0.034,Y -527.027,Z 1178.432,A 0.000,B 0.000,C 90.000,E1 293.695} C_DIS
LIN {X 0.017,Y -526.806,Z 1178.420,A 0.000,B 0.000,C 90.000,E1 291.663} C_DIS
LIN {X -0.108,Y -526.526,Z 1178.411,A 0.000,B 0.000,C 90.000,E1 289.939} C_DIS
LIN {X 0.238,Y -526.124,Z 1178.400,A 0.000,B 0.000,C 90.000,E1 287.873} C_DIS
LIN {X 0.072,Y -525.727,Z 1178.393,A 0.000,B 0.000,C 90.000,E1 286.732} C_DIS
LIN {X -0.073,Y -524.713,Z 1178.382,A 0.000,B 0.000,C 90.000,E1 284.717} C_DIS
LIN {X 0.107,Y -523.980,Z 1178.375,A 0.000,B 0.000,C 90.000,E1 283.536} C_DIS
LIN {X -0.201,Y -522.348,Z 1178.362,A 0.000,B 0.000,C 90.000,E1 281.243} C_DIS
LIN {X -0.253,Y -521.180,Z 1178.351,A 0.000,B 0.000,C 90.000,E1 279.208} C_DIS
LIN {X 0.178,Y -520.156,Z 1178.341,A 0.000,B 0.000,C 90.000,E1 277.409} C_DIS
LIN {X -0.065,Y -519.056,Z 1178.332,A 0.000,B 0.000,C 90.000,E1 275.682} C_DIS
LIN {X 0.212,Y -518.173,Z 1178.323,A 0.000,B 0.000,C 90.000,E1 274.188} C_DIS
LIN {X -0.174,Y -517.110,Z 1178.312,A 0.000,B 0.000,C 90.000,E1 272.178} C_DIS
LIN {X -0.028,Y -516.308,Z 1178.302,A 0.000,B 0.000,C 90.000,E1 270.401} C_DIS
LIN {X 0.017,Y -515.355,Z 1178.291,A 0.000,B 0.000,C 90.000,E1 268.339} C_DIS
LIN {X -0.252,Y -514.813,Z 1178.284,A 0.000,B 0.000,C 90.000,E1 267.192} C_DIS
LIN {X -0.057,Y -513.825,Z 1178.276,A 0.000,B 0.000,C 90.000,E1 265.698} C_DIS
LIN {X 0.119,Y -512.579,Z 1178.268,A 0.000,B 0.000,C 90.000,E1 264.204} C_DIS
LIN {X -0.150,Y -511.620,Z 1178.261,A 0.000,B 0.000,C 90.000,E1 263.053} C_DIS
LIN {X 0.136,Y -510.470,Z 1178.255,A 0.000,B 0.000,C 90.000,E1 261.837} C_DIS
LIN {X -0.140,Y -509.136,Z 1178.247,A 0.000,B 0.000,C 90.000,E1 260.387} C_DIS
LIN {X 0.016,Y -507.058,Z 1178.233,A 0.000,B 0.000,C 90.000,E1 257.993} C_DIS
LIN {X -0.227,Y -505.341,Z 1178.222,A 0.000,B 0.000,C 90.000,E1 255.936} C_DIS
LIN {X 0.154,Y -503.255,Z 1178.208,A 0.000,B 0.000,C 90.000,E1 253.504} C_DIS
LIN {X 0.144,Y -502.241,Z 1178.202,A 0.000,B 0.000,C 90.000,E1 252.308} C_DIS
LIN {X 0.204,Y -501.543,Z 1178.197,A 0.000,B 0.000,C 90.000,E1 251.402} C_DIS
LIN {X -0.075,Y -500.241,Z 1178.188,A 0.000,B 0.000,C 90.000,E1 249.934} C_DIS
LIN {X 0.093,Y -498.772,Z 1178.180,A 0.000,B 0.000,C 90.000,E1 248.411} C_DIS
LIN {X -0.051,Y -497.337,Z 1178.172,A 0.000,B 0.000,C 90.000,E1 246.922} C_DIS
LIN {X -0.022,Y -495.738,Z 1178.163,A 0.000,B 0.000,C 90.000,E1 245.409} C_DIS
LIN {X -0.022,Y -493.999,Z 1178.155,A 0.000,B 0.000,C 90.000,E1 243.896} C_DIS
LIN {X 0.155,Y -492.021,Z 1178.147,A 0.000,B 0.000,C 90.000,E1 242.359} C_DIS
LIN {X -0.077,Y -489.212,Z 1178.135,A 0.000,B 0.000,C 90.000,E1 240.255} C_DIS
LIN {X -0.192,Y -487.128,Z 1178.126,A 0.000,B 0.000,C 90.000,E1 238.742} C_DIS
LIN {X 0.158,Y -484.969,Z 1178.118,A 0.000,B 0.000,C 90.000,E1 237.168} C_DIS
LIN {X -0.083,Y -481.533,Z 1178.104,A 0.000,B 0.000,C 90.000,E1 234.736} C_DIS
LIN {X -0.242,Y -479.444,Z 1178.095,A 0.000,B 0.000,C 90.000,E1 233.210} C_DIS
LIN {X -0.186,Y -475.998,Z 1178.082,A 0.000,B 0.000,C 90.000,E1 230.723} C_DIS
LIN {X -0.169,Y -473.634,Z 1178.071,A 0.000,B 0.000,C 90.000,E1 228.852} C_DIS
LIN {X -0.202,Y -472.301,Z 1178.066,A 0.000,B 0.000,C 90.000,E1 227.919} C_DIS
LIN {X 0.081,Y -467.364,Z 1178.047,A 0.000,B 0.000,C 90.000,E1 224.433} C_DIS
LIN {X 0.047,Y -464.435,Z 1178.031,A 0.000,B 0.000,C 90.000,E1 221.595} C_DIS
LIN {X -0.249,Y -462.891,Z 1178.014,A 0.000,B 0.000,C 90.000,E1 218.463} C_DIS
LIN {X -0.198,Y -462.551,Z 1178.005,A 0.000,B 0.000,C 90.000,E1 216.870} C_DIS
LIN {X -0.022,Y -462.737,Z 1177.978,A 0.000,B 0.000,C 90.000,E1 212.084} C_DIS
LIN {X 0.044,Y -464.371,Z 1177.964,A 0.000,B 0.000,C 90.000,E1 209.539} C_DIS
LIN {X -0.106,Y -465.728,Z 1177.955,A 0.000,B 0.000,C 90.000,E1 207.975} C_DIS
LIN {X -0.277,Y -468.653,Z 1177.940,A 0.000,B 0.000,C 90.000,E1 205.155} C_DIS
LIN {X -0.056,Y -476.317,Z 1177.913,A 0.000,B 0.000,C 90.000,E1 200.429} C_DIS
LIN {X -0.216,Y -484.314,Z 1177.895,A 0.000,B 0.000,C 90.000,E1 197.040} C_DIS
LIN {X 0.003,Y -493.312,Z 1177.878,A 0.000,B 0.000,C 90.000,E1 193.953} C_DIS
LIN {X 0.070,Y -500.088,Z 1177.866,A 0.000,B 0.000,C 90.000,E1 191.827} C_DIS
LIN {X 0.213,Y -505.114,Z 1177.857,A 0.000,B 0.000,C 90.000,E1 190.310} C_DIS
LIN {X 0.177,Y -513.331,Z 1177.844,A 0.000,B 0.000,C 90.000,E1 187.936} C_DIS
LIN {X -0.005,Y -517.520,Z 1177.838,A 0.000,B 0.000,C 90.000,E1 186.777} C_DIS
LIN {X -0.193,Y -521.522,Z 1177.831,A 0.000,B 0.000,C 90.000,E1 185.625} C_DIS
LIN {X 0.155,Y -527.631,Z 1177.822,A 0.000,B 0.000,C 90.000,E1 183.841} C_DIS
LIN {X 0.044,Y -533.738,Z 1177.812,A 0.000,B 0.000,C 90.000,E1 182.121} C_DIS
LIN {X 0.101,Y -541.703,Z 1177.799,A 0.000,B 0.000,C 90.000,E1 179.828} C_DIS
LIN {X 0.246,Y -546.747,Z 1177.791,A 0.000,B 0.000,C 90.000,E1 178.396} C_DIS
LIN {X 0.030,Y -552.662,Z 1177.782,A 0.000,B 0.000,C 90.000,E1 176.731} C_DIS
LIN {X -0.054,Y -558.517,Z 1177.773,A 0.000,B 0.000,C 90.000,E1 175.065} C_DIS
LIN {X 0.036,Y -564.328,Z 1177.763,A 0.000,B 0.000,C 90.000,E1 173.394} C_DIS
LIN {X 0.241,Y -570.029,Z 1177.754,A 0.000,B 0.000,C 90.000,E1 171.724} C_DIS
LIN {X -0.038,Y -574.786,Z 1177.747,A 0.000,B 0.000,C 90.000,E1 170.387} C_DIS
LIN {X -0.235,Y -579.407,Z 1177.739,A 0.000,B 0.000,C 90.000,E1 169.050} C_DIS
LIN {X -0.242,Y -583.974,Z 1177.732,A 0.000,B 0.000,C 90.000,E1 167.701} C_DIS
LIN {X -0.168,Y -588.573,Z 1177.724,A 0.000,B 0.000,C 90.000,E1 166.353} C_DIS
LIN {X 0.124,Y -592.943,Z 1177.717,A 0.000,B 0.000,C 90.000,E1 164.991} C_DIS
LIN {X -0.081,Y -597.318,Z 1177.709,A 0.000,B 0.000,C 90.000,E1 163.685} C_DIS
LIN {X 0.245,Y -600.743,Z 1177.703,A 0.000,B 0.000,C 90.000,E1 162.598} C_DIS
LIN {X -0.136,Y -604.100,Z 1177.698,A 0.000,B 0.000,C 90.000,E1 161.583} C_DIS
LIN {X 0.216,Y -608.148,Z 1177.690,A 0.000,B 0.000,C 90.000,E1 160.242} C_DIS
LIN {X 0.073,Y -612.062,Z 1177.683,A 0.000,B 0.000,C 90.000,E1 158.954} C_DIS
LIN {X -0.006,Y -615.834,Z 1177.676,A 0.000,B 0.000,C 90.000,E1 157.667} C_DIS
LIN {X 0.208,Y -619.601,Z 1177.669,A 0.000,B 0.000,C 90.000,E1 156.357} C_DIS
LIN {X -0.079,Y -622.555,Z 1177.663,A 0.000,B 0.000,C 90.000,E1 155.357} C_DIS
LIN {X -0.053,Y -625.996,Z 1177.656,A 0.000,B 0.000,C 90.000,E1 154.076} C_DIS
LIN {X 0.037,Y -629.462,Z 1177.649,A 0.000,B 0.000,C 90.000,E1 152.794} C_DIS
LIN {X 0.211,Y -633.436,Z 1177.641,A 0.000,B 0.000,C 90.000,E1 151.257} C_DIS
LIN {X 0.120,Y -635.941,Z 1177.635,A 0.000,B 0.000,C 90.000,E1 150.255} C_DIS
LIN {X 0.069,Y -638.378,Z 1177.629,A 0.000,B 0.000,C 90.000,E1 149.253} C_DIS
LIN {X 0.152,Y -641.724,Z 1177.621,A 0.000,B 0.000,C 90.000,E1 147.740} C_DIS
LIN {X -0.025,Y -643.767,Z 1177.615,A 0.000,B 0.000,C 90.000,E1 146.755} C_DIS
LIN {X -0.105,Y -646.177,Z 1177.608,A 0.000,B 0.000,C 90.000,E1 145.515} C_DIS
LIN {X -0.155,Y -648.460,Z 1177.602,A 0.000,B 0.000,C 90.000,E1 144.276} C_DIS
LIN {X 0.201,Y -650.663,Z 1177.595,A 0.000,B 0.000,C 90.000,E1 143.004} C_DIS
LIN {X 0.072,Y -652.828,Z 1177.588,A 0.000,B 0.000,C 90.000,E1 141.778} C_DIS
LIN {X -0.068,Y -654.617,Z 1177.582,A 0.000,B 0.000,C 90.000,E1 140.803} C_DIS
LIN {X -0.228,Y -658.007,Z 1177.573,A 0.000,B 0.000,C 90.000,E1 139.094} C_DIS
LIN {X 0.091,Y -661.159,Z 1177.564,A 0.000,B 0.000,C 90.000,E1 137.595} C_DIS
LIN {X 0.031,Y -664.211,Z 1177.556,A 0.000,B 0.000,C 90.000,E1 136.134} C_DIS
LIN {X 0.020,Y -669.489,Z 1177.543,A 0.000,B 0.000,C 90.000,E1 133.704} C_DIS
LIN {X 0.159,Y -674.097,Z 1177.532,A 0.000,B 0.000,C 90.000,E1 131.757} C_DIS
LIN {X -0.448,Y -679.240,Z 1177.520,A 0.000,B 0.000,C 90.000,E1 129.644} C_DIS
LIN {X -0.240,Y -681.666,Z 1177.515,A 0.000,B 0.000,C 90.000,E1 128.669} C_DIS
LIN {X -0.206,Y -685.843,Z 1177.505,A 0.000,B 0.000,C 90.000,E1 126.996} C_DIS
LIN {X 0.432,Y -689.396,Z 1177.498,A 0.000,B 0.000,C 90.000,E1 125.518} C_DIS
LIN {X -0.421,Y -692.277,Z 1177.491,A 0.000,B 0.000,C 90.000,E1 124.405} C_DIS
LIN {X 0.078,Y -694.390,Z 1177.486,A 0.000,B 0.000,C 90.000,E1 123.420} C_DIS
LIN {X -0.129,Y -696.982,Z 1177.479,A 0.000,B 0.000,C 90.000,E1 122.260} C_DIS
LIN {X -0.323,Y -698.911,Z 1177.474,A 0.000,B 0.000,C 90.000,E1 121.337} C_DIS
LIN {X -0.129,Y -700.739,Z 1177.469,A 0.000,B 0.000,C 90.000,E1 120.384} C_DIS
LIN {X 0.068,Y -701.944,Z 1177.465,A 0.000,B 0.000,C 90.000,E1 119.667} C_DIS
LIN {X 0.223,Y -703.886,Z 1177.458,A 0.000,B 0.000,C 90.000,E1 118.487} C_DIS
LIN {X -0.212,Y -705.311,Z 1177.453,A 0.000,B 0.000,C 90.000,E1 117.590} C_DIS
LIN {X 0.033,Y -706.088,Z 1177.449,A 0.000,B 0.000,C 90.000,E1 116.873} C_DIS
LIN {X -0.374,Y -706.587,Z 1177.444,A 0.000,B 0.000,C 90.000,E1 115.976} C_DIS
LIN {X 0.214,Y -706.711,Z 1177.442,A 0.000,B 0.000,C 90.000,E1 115.463} C_DIS
LIN {X -0.138,Y -706.697,Z 1177.439,A 0.000,B 0.000,C 90.000,E1 115.027} C_DIS
LIN {X -0.193,Y -706.423,Z 1177.436,A 0.000,B 0.000,C 90.000,E1 114.567} C_DIS
LIN {X 0.098,Y -705.565,Z 1177.434,A 0.000,B 0.000,C 90.000,E1 114.079} C_DIS
LIN {X 0.386,Y -704.988,Z 1177.433,A 0.000,B 0.000,C 90.000,E1 113.823} C_DIS
LIN {X 0.029,Y -702.961,Z 1177.430,A 0.000,B 0.000,C 90.000,E1 113.387} C_DIS
LIN {X 0.169,Y -702.358,Z 1177.429,A 0.000,B 0.000,C 90.000,E1 113.259} C_DIS
LIN {X 0.032,Y -701.441,Z 1177.429,A 0.000,B 0.000,C 90.000,E1 113.153} C_DIS
LIN {X -0.130,Y -696.673,Z 1177.426,A 0.000,B 0.000,C 90.000,E1 112.717} C_DIS
LIN {X 0.054,Y -695.088,Z 1177.426,A 0.000,B 0.000,C 90.000,E1 112.589} C_DIS
LIN {X 0.235,Y -692.238,Z 1177.425,A 0.000,B 0.000,C 90.000,E1 112.461} C_DIS
LIN {X 0.194,Y -686.183,Z 1177.424,A 0.000,B 0.000,C 90.000,E1 112.280} C_DIS
LIN {X -0.120,Y -684.990,Z 1177.424,A 0.000,B 0.000,C 90.000,E1 112.280} C_DIS
LIN {X -0.276,Y -683.803,Z 1177.424,A 0.000,B 0.000,C 90.000,E1 112.280} C_DIS
LIN {X 0.256,Y -676.593,Z 1177.424,A 0.000,B 0.000,C 90.000,E1 112.206} C_DIS
LIN {X 0.188,Y -605.512,Z 1177.423,A 0.000,B 0.000,C 90.000,E1 112.206} C_DIS
LIN {X 0.251,Y -600.977,Z 1177.422,A 0.000,B 0.000,C 90.000,E1 111.897} C_DIS
LIN {X -0.136,Y -592.804,Z 1177.418,A 0.000,B 0.000,C 90.000,E1 111.280} C_DIS
LIN {X -0.266,Y -584.647,Z 1177.414,A 0.000,B 0.000,C 90.000,E1 110.610} C_DIS
LIN {X 0.027,Y -576.109,Z 1177.411,A 0.000,B 0.000,C 90.000,E1 109.885} C_DIS
LIN {X -0.329,Y -571.525,Z 1177.409,A 0.000,B 0.000,C 90.000,E1 109.577} C_DIS
LIN {X 0.135,Y -562.737,Z 1177.405,A 0.000,B 0.000,C 90.000,E1 108.906} C_DIS
LIN {X 0.000,Y -555.741,Z 1177.402,A 0.000,B 0.000,C 90.000,E1 108.417} C_DIS
LIN {X -0.152,Y -552.150,Z 1177.401,A 0.000,B 0.000,C 90.000,E1 108.109} C_DIS
LIN {X -0.200,Y -550.912,Z 1177.399,A 0.000,B 0.000,C 90.000,E1 107.873} C_DIS
LIN {X -0.247,Y -550.284,Z 1177.397,A 0.000,B 0.000,C 90.000,E1 107.457} C_DIS
LIN {X 0.228,Y -550.511,Z 1177.393,A 0.000,B 0.000,C 90.000,E1 106.677} C_DIS
LIN {X 0.041,Y -552.783,Z 1177.379,A 0.000,B 0.000,C 90.000,E1 104.175} C_DIS
LIN {X 0.227,Y -554.218,Z 1177.370,A 0.000,B 0.000,C 90.000,E1 102.479} C_DIS
LIN {X 0.179,Y -556.562,Z 1177.357,A 0.000,B 0.000,C 90.000,E1 100.254} C_DIS
LIN {X -0.145,Y -558.525,Z 1177.346,A 0.000,B 0.000,C 90.000,E1 98.341} C_DIS
LIN {X -0.083,Y -559.728,Z 1177.339,A 0.000,B 0.000,C 90.000,E1 96.947} C_DIS
LIN {X -0.217,Y -560.622,Z 1177.332,A 0.000,B 0.000,C 90.000,E1 95.853} C_DIS
LIN {X -0.032,Y -561.898,Z 1177.322,A 0.000,B 0.000,C 90.000,E1 93.898} C_DIS
LIN {X -0.216,Y -563.745,Z 1177.308,A 0.000,B 0.000,C 90.000,E1 91.432} C_DIS
LIN {X -0.245,Y -564.756,Z 1177.300,A 0.000,B 0.000,C 90.000,E1 90.057} C_DIS
LIN {X -0.144,Y -565.918,Z 1177.291,A 0.000,B 0.000,C 90.000,E1 88.396} C_DIS
LIN {X 0.021,Y -566.990,Z 1177.282,A 0.000,B 0.000,C 90.000,E1 86.731} C_DIS
LIN {X -0.235,Y -568.254,Z 1177.271,A 0.000,B 0.000,C 90.000,E1 84.837} C_DIS
LIN {X -0.075,Y -569.187,Z 1177.264,A 0.000,B 0.000,C 90.000,E1 83.451} C_DIS
LIN {X 0.109,Y -570.162,Z 1177.256,A 0.000,B 0.000,C 90.000,E1 82.064} C_DIS
LIN {X -0.264,Y -570.937,Z 1177.248,A 0.000,B 0.000,C 90.000,E1 80.735} C_DIS
LIN {X -0.152,Y -571.987,Z 1177.238,A 0.000,B 0.000,C 90.000,E1 78.814} C_DIS
LIN {X -0.100,Y -572.808,Z 1177.229,A 0.000,B 0.000,C 90.000,E1 77.173} C_DIS
LIN {X 0.100,Y -573.668,Z 1177.220,A 0.000,B 0.000,C 90.000,E1 75.519} C_DIS
LIN {X -0.075,Y -574.221,Z 1177.214,A 0.000,B 0.000,C 90.000,E1 74.448} C_DIS
LIN {X 0.310,Y -575.392,Z 1177.202,A 0.000,B 0.000,C 90.000,E1 72.236} C_DIS
LIN {X 0.339,Y -576.401,Z 1177.193,A 0.000,B 0.000,C 90.000,E1 70.604} C_DIS
LIN {X 0.202,Y -577.342,Z 1177.185,A 0.000,B 0.000,C 90.000,E1 69.263} C_DIS
LIN {X 0.026,Y -580.136,Z 1177.168,A 0.000,B 0.000,C 90.000,E1 66.305} C_DIS
LIN {X 0.133,Y -580.895,Z 1177.164,A 0.000,B 0.000,C 90.000,E1 65.485} C_DIS
LIN {X -0.150,Y -582.407,Z 1177.155,A 0.000,B 0.000,C 90.000,E1 63.896} C_DIS
LIN {X -0.140,Y -583.943,Z 1177.146,A 0.000,B 0.000,C 90.000,E1 62.281} C_DIS
LIN {X -0.100,Y -585.499,Z 1177.137,A 0.000,B 0.000,C 90.000,E1 60.667} C_DIS
LIN {X -0.136,Y -586.618,Z 1177.130,A 0.000,B 0.000,C 90.000,E1 59.331} C_DIS
LIN {X -0.149,Y -587.710,Z 1177.122,A 0.000,B 0.000,C 90.000,E1 57.995} C_DIS
LIN {X 0.233,Y -589.079,Z 1177.112,A 0.000,B 0.000,C 90.000,E1 56.087} C_DIS
LIN {X 0.285,Y -590.140,Z 1177.103,A 0.000,B 0.000,C 90.000,E1 54.482} C_DIS
LIN {X -0.332,Y -591.037,Z 1177.095,A 0.000,B 0.000,C 90.000,E1 53.210} C_DIS
LIN {X 0.050,Y -592.322,Z 1177.084,A 0.000,B 0.000,C 90.000,E1 51.045} C_DIS
LIN {X 0.192,Y -592.990,Z 1177.076,A 0.000,B 0.000,C 90.000,E1 49.703} C_DIS
LIN {X -0.104,Y -593.453,Z 1177.069,A 0.000,B 0.000,C 90.000,E1 48.405} C_DIS
LIN {X 0.008,Y -593.741,Z 1177.062,A 0.000,B 0.000,C 90.000,E1 47.067} C_DIS
LIN {X -0.251,Y -593.849,Z 1177.057,A 0.000,B 0.000,C 90.000,E1 46.296} C_DIS
LIN {X 0.052,Y -593.638,Z 1177.048,A 0.000,B 0.000,C 90.000,E1 44.676} C_DIS
LIN {X -0.029,Y -593.271,Z 1177.042,A 0.000,B 0.000,C 90.000,E1 43.623} C_DIS
LIN {X 0.311,Y -592.682,Z 1177.036,A 0.000,B 0.000,C 90.000,E1 42.528} C_DIS
LIN {X -0.196,Y -592.014,Z 1177.031,A 0.000,B 0.000,C 90.000,E1 41.515} C_DIS
LIN {X -0.026,Y -591.406,Z 1177.026,A 0.000,B 0.000,C 90.000,E1 40.701} C_DIS
LIN {X 0.100,Y -590.080,Z 1177.019,A 0.000,B 0.000,C 90.000,E1 39.358} C_DIS
LIN {X -0.003,Y -588.831,Z 1177.013,A 0.000,B 0.000,C 90.000,E1 38.302} C_DIS
LIN {X -0.028,Y -587.422,Z 1177.007,A 0.000,B 0.000,C 90.000,E1 37.237} C_DIS
LIN {X 0.089,Y -586.137,Z 1177.002,A 0.000,B 0.000,C 90.000,E1 36.423} C_DIS
LIN {X -0.128,Y -583.561,Z 1176.995,A 0.000,B 0.000,C 90.000,E1 35.105} C_DIS
LIN {X 0.252,Y -580.965,Z 1176.989,A 0.000,B 0.000,C 90.000,E1 33.992} C_DIS
LIN {X -0.054,Y -578.688,Z 1176.984,A 0.000,B 0.000,C 90.000,E1 33.214} C_DIS
LIN {X -0.067,Y -575.034,Z 1176.979,A 0.000,B 0.000,C 90.000,E1 32.133} C_DIS
LIN {X -0.257,Y -571.945,Z 1176.974,A 0.000,B 0.000,C 90.000,E1 31.337} C_DIS
LIN {X 0.101,Y -568.989,Z 1176.970,A 0.000,B 0.000,C 90.000,E1 30.620} C_DIS
LIN {X 0.133,Y -565.080,Z 1176.966,A 0.000,B 0.000,C 90.000,E1 29.795} C_DIS
LIN {X -0.149,Y -562.938,Z 1176.963,A 0.000,B 0.000,C 90.000,E1 29.411} C_DIS
LIN {X -0.079,Y -557.584,Z 1176.958,A 0.000,B 0.000,C 90.000,E1 28.437} C_DIS
LIN {X 0.036,Y -552.583,Z 1176.953,A 0.000,B 0.000,C 90.000,E1 27.590} C_DIS
LIN {X -0.046,Y -549.916,Z 1176.951,A 0.000,B 0.000,C 90.000,E1 27.180} C_DIS
LIN {X -0.148,Y -545.024,Z 1176.947,A 0.000,B 0.000,C 90.000,E1 26.488} C_DIS
LIN {X -0.048,Y -539.854,Z 1176.943,A 0.000,B 0.000,C 90.000,E1 25.771} C_DIS
LIN {X 0.252,Y -534.289,Z 1176.939,A 0.000,B 0.000,C 90.000,E1 25.027} C_DIS
LIN {X 0.049,Y -524.398,Z 1176.933,A 0.000,B 0.000,C 90.000,E1 23.898} C_DIS
LIN {X -0.056,Y -519.213,Z 1176.930,A 0.000,B 0.000,C 90.000,E1 23.334} C_DIS
LIN {X -0.135,Y -512.534,Z 1176.926,A 0.000,B 0.000,C 90.000,E1 22.642} C_DIS
LIN {X -0.157,Y -505.753,Z 1176.922,A 0.000,B 0.000,C 90.000,E1 21.950} C_DIS
LIN {X 0.158,Y -498.719,Z 1176.918,A 0.000,B 0.000,C 90.000,E1 21.227} C_DIS
LIN {X 0.060,Y -488.711,Z 1176.913,A 0.000,B 0.000,C 90.000,E1 20.301} C_DIS
LIN {X -0.116,Y -476.968,Z 1176.907,A 0.000,B 0.000,C 90.000,E1 19.268} C_DIS
LIN {X 0.167,Y -469.856,Z 1176.903,A 0.000,B 0.000,C 90.000,E1 18.598} C_DIS
LIN {X -0.154,Y -459.994,Z 1176.899,A 0.000,B 0.000,C 90.000,E1 17.764} C_DIS
LIN {X 0.217,Y -438.182,Z 1176.887,A 0.000,B 0.000,C 90.000,E1 15.662} C_DIS
LIN {X 0.114,Y -425.302,Z 1176.880,A 0.000,B 0.000,C 90.000,E1 14.356} C_DIS
LIN {X -0.018,Y -414.151,Z 1176.873,A 0.000,B 0.000,C 90.000,E1 13.119} C_DIS
LIN {X 0.053,Y -402.043,Z 1176.865,A 0.000,B 0.000,C 90.000,E1 11.591} C_DIS
LIN {X 0.039,Y -397.200,Z 1176.861,A 0.000,B 0.000,C 90.000,E1 10.894} C_DIS
LIN {X 0.040,Y -394.317,Z 1176.858,A 0.000,B 0.000,C 90.000,E1 10.366} C_DIS
LIN {X 0.112,Y -393.033,Z 1176.855,A 0.000,B 0.000,C 90.000,E1 9.962} C_DIS
LIN {X -0.116,Y -392.937,Z 1176.855,A 0.000,B 0.000,C 90.000,E1 9.962} C_DIS
LIN {X -0.154,Y -392.940,Z 1176.855,A 0.000,B 0.000,C 90.000,E1 9.962} C_DIS
LIN {X -0.063,Y -393.301,Z 1176.853,A 0.000,B 0.000,C 90.000,E1 9.500} C_DIS
LIN {X -0.143,Y -394.962,Z 1176.849,A 0.000,B 0.000,C 90.000,E1 8.803} C_DIS
LIN {X 0.196,Y -398.323,Z 1176.844,A 0.000,B 0.000,C 90.000,E1 7.871} C_DIS
LIN {X -0.206,Y -402.152,Z 1176.839,A 0.000,B 0.000,C 90.000,E1 7.125} C_DIS
LIN {X -0.066,Y -406.318,Z 1176.836,A 0.000,B 0.000,C 90.000,E1 6.543} C_DIS
LIN {X -0.091,Y -407.926,Z 1176.835,A 0.000,B 0.000,C 90.000,E1 6.372} C_DIS
LIN {X 0.026,Y -413.110,Z 1176.833,A 0.000,B 0.000,C 90.000,E1 5.910} C_DIS
LIN {X 0.030,Y -430.360,Z 1176.826,A 0.000,B 0.000,C 90.000,E1 4.588} C_DIS
LIN {X 0.173,Y -449.659,Z 1176.818,A 0.000,B 0.000,C 90.000,E1 3.154} C_DIS
LIN {X -0.099,Y -462.327,Z 1176.813,A 0.000,B 0.000,C 90.000,E1 2.293} C_DIS
LIN {X 0.052,Y -471.645,Z 1176.809,A 0.000,B 0.000,C 90.000,E1 1.604} C_DIS
LIN {X -0.033,Y -480.964,Z 1176.805,A 0.000,B 0.000,C 90.000,E1 0.917} C_DIS
LIN {X -0.101,Y -485.508,Z 1176.803,A 0.000,B 0.000,C 90.000,E1 0.573} C_DIS
LIN {X 0.140,Y -491.487,Z 1176.800,A 0.000,B 0.000,C 90.000,E1 0.057} C_DIS
LIN {X -0.035,Y -497.648,Z 1176.797,A 0.000,B 0.000,C 90.000,E1 359.542} C_DIS
LIN {X -0.153,Y -503.279,Z 1176.795,A 0.000,B 0.000,C 90.000,E1 359.026} C_DIS
LIN {X 0.134,Y -511.165,Z 1176.790,A 0.000,B 0.000,C 90.000,E1 358.165} C_DIS
LIN {X -0.186,Y -517.468,Z 1176.786,A 0.000,B 0.000,C 90.000,E1 357.478} C_DIS
LIN {X 0.159,Y -523.213,Z 1176.782,A 0.000,B 0.000,C 90.000,E1 356.731} C_DIS
LIN {X -0.214,Y -528.509,Z 1176.778,A 0.000,B 0.000,C 90.000,E1 356.045} C_DIS
LIN {X 0.015,Y -533.383,Z 1176.774,A 0.000,B 0.000,C 90.000,E1 355.298} C_DIS
LIN {X 0.031,Y -536.930,Z 1176.771,A 0.000,B 0.000,C 90.000,E1 354.723} C_DIS
LIN {X -0.194,Y -540.919,Z 1176.767,A 0.000,B 0.000,C 90.000,E1 354.033} C_DIS
LIN {X -0.063,Y -543.834,Z 1176.764,A 0.000,B 0.000,C 90.000,E1 353.451} C_DIS
LIN {X -0.230,Y -547.162,Z 1176.760,A 0.000,B 0.000,C 90.000,E1 352.761} C_DIS
LIN {X -0.115,Y -549.622,Z 1176.757,A 0.000,B 0.000,C 90.000,E1 352.186} C_DIS
LIN {X 0.092,Y -551.935,Z 1176.753,A 0.000,B 0.000,C 90.000,E1 351.602} C_DIS
LIN {X -0.191,Y -554.993,Z 1176.749,A 0.000,B 0.000,C 90.000,E1 350.792} C_DIS
LIN {X 0.099,Y -557.766,Z 1176.744,A 0.000,B 0.000,C 90.000,E1 349.926} C_DIS
LIN {X -0.032,Y -560.297,Z 1176.740,A 0.000,B 0.000,C 90.000,E1 349.106} C_DIS
LIN {X 0.023,Y -563.357,Z 1176.733,A 0.000,B 0.000,C 90.000,E1 347.993} C_DIS
LIN {X -0.261,Y -566.870,Z 1176.726,A 0.000,B 0.000,C 90.000,E1 346.645} C_DIS
LIN {X 0.196,Y -570.069,Z 1176.718,A 0.000,B 0.000,C 90.000,E1 345.227} C_DIS
LIN {X -0.030,Y -572.487,Z 1176.712,A 0.000,B 0.000,C 90.000,E1 344.157} C_DIS
LIN {X -0.228,Y -575.864,Z 1176.703,A 0.000,B 0.000,C 90.000,E1 342.543} C_DIS
LIN {X 0.170,Y -578.459,Z 1176.695,A 0.000,B 0.000,C 90.000,E1 341.148} C_DIS
LIN {X 0.231,Y -580.264,Z 1176.689,A 0.000,B 0.000,C 90.000,E1 340.061} C_DIS
LIN {X -0.238,Y -581.922,Z 1176.683,A 0.000,B 0.000,C 90.000,E1 339.028} C_DIS
LIN {X -0.075,Y -583.562,Z 1176.676,A 0.000,B 0.000,C 90.000,E1 337.667} C_DIS
LIN {X -0.161,Y -584.209,Z 1176.672,A 0.000,B 0.000,C 90.000,E1 336.869} C_DIS
LIN {X -0.139,Y -584.646,Z 1176.666,A 0.000,B 0.000,C 90.000,E1 335.793} C_DIS
LIN {X 0.144,Y -584.625,Z 1176.662,A 0.000,B 0.000,C 90.000,E1 335.229} C_DIS
LIN {X 0.177,Y -584.130,Z 1176.656,A 0.000,B 0.000,C 90.000,E1 334.152} C_DIS
LIN {X -0.198,Y -583.447,Z 1176.652,A 0.000,B 0.000,C 90.000,E1 333.384} C_DIS
LIN {X 0.207,Y -582.273,Z 1176.648,A 0.000,B 0.000,C 90.000,E1 332.538} C_DIS
LIN {X -0.185,Y -580.828,Z 1176.643,A 0.000,B 0.000,C 90.000,E1 331.769} C_DIS
LIN {X 0.191,Y -579.004,Z 1176.639,A 0.000,B 0.000,C 90.000,E1 330.923} C_DIS
LIN {X 0.041,Y -576.845,Z 1176.634,A 0.000,B 0.000,C 90.000,E1 330.127} C_DIS
LIN {X -0.109,Y -576.006,Z 1176.633,A 0.000,B 0.000,C 90.000,E1 329.871} C_DIS
LIN {X -0.128,Y -574.064,Z 1176.630,A 0.000,B 0.000,C 90.000,E1 329.331} C_DIS
LIN {X -0.075,Y -572.377,Z 1176.627,A 0.000,B 0.000,C 90.000,E1 328.918} C_DIS
LIN {X 0.187,Y -568.101,Z 1176.623,A 0.000,B 0.000,C 90.000,E1 328.074} C_DIS
LIN {X 0.110,Y -564.925,Z 1176.620,A 0.000,B 0.000,C 90.000,E1 327.533} C_DIS
LIN {X 0.211,Y -560.319,Z 1176.616,A 0.000,B 0.000,C 90.000,E1 326.834} C_DIS
LIN {X 0.181,Y -556.480,Z 1176.613,A 0.000,B 0.000,C 90.000,E1 326.294} C_DIS
LIN {X 0.021,Y -552.170,Z 1176.610,A 0.000,B 0.000,C 90.000,E1 325.754} C_DIS
LIN {X 0.192,Y -545.256,Z 1176.605,A 0.000,B 0.000,C 90.000,E1 324.895} C_DIS
LIN {X 0.123,Y -539.071,Z 1176.601,A 0.000,B 0.000,C 90.000,E1 324.196} C_DIS
LIN {X 0.233,Y -523.968,Z 1176.592,A 0.000,B 0.000,C 90.000,E1 322.477} C_DIS
LIN {X 0.059,Y -520.375,Z 1176.589,A 0.000,B 0.000,C 90.000,E1 321.984} C_DIS
LIN {X 0.145,Y -517.985,Z 1176.586,A 0.000,B 0.000,C 90.000,E1 321.537} C_DIS
LIN {X 0.023,Y -516.091,Z 1176.583,A 0.000,B 0.000,C 90.000,E1 320.964} C_DIS
LIN {X 0.216,Y -515.259,Z 1176.579,A 0.000,B 0.000,C 90.000,E1 320.194} C_DIS
LIN {X 0.070,Y -515.209,Z 1176.576,A 0.000,B 0.000,C 90.000,E1 319.622} C_DIS
LIN {X -0.101,Y -516.159,Z 1176.566,A 0.000,B 0.000,C 90.000,E1 317.877} C_DIS
LIN {X 0.268,Y -517.493,Z 1176.553,A 0.000,B 0.000,C 90.000,E1 315.486} C_DIS
LIN {X 0.201,Y -518.359,Z 1176.545,A 0.000,B 0.000,C 90.000,E1 314.028} C_DIS
LIN {X 0.068,Y -519.356,Z 1176.535,A 0.000,B 0.000,C 90.000,E1 312.285} C_DIS
LIN {X 0.050,Y -520.286,Z 1176.527,A 0.000,B 0.000,C 90.000,E1 310.825} C_DIS
LIN {X 0.110,Y -521.206,Z 1176.519,A 0.000,B 0.000,C 90.000,E1 309.358} C_DIS
LIN {X 0.151,Y -522.309,Z 1176.509,A 0.000,B 0.000,C 90.000,E1 307.604} C_DIS
LIN {X -0.106,Y -523.273,Z 1176.499,A 0.000,B 0.000,C 90.000,E1 305.884} C_DIS
LIN {X 0.033,Y -524.405,Z 1176.488,A 0.000,B 0.000,C 90.000,E1 303.833} C_DIS
LIN {X -0.311,Y -525.239,Z 1176.480,A 0.000,B 0.000,C 90.000,E1 302.418} C_DIS
LIN {X -0.230,Y -526.140,Z 1176.470,A 0.000,B 0.000,C 90.000,E1 300.669} C_DIS
LIN {X -0.038,Y -526.597,Z 1176.464,A 0.000,B 0.000,C 90.000,E1 299.489} C_DIS
LIN {X 0.106,Y -527.042,Z 1176.456,A 0.000,B 0.000,C 90.000,E1 298.025} C_DIS
LIN {X -0.246,Y -527.284,Z 1176.448,A 0.000,B 0.000,C 90.000,E1 296.616} C_DIS
LIN {X -0.115,Y -527.457,Z 1176.440,A 0.000,B 0.000,C 90.000,E1 295.155} C_DIS
